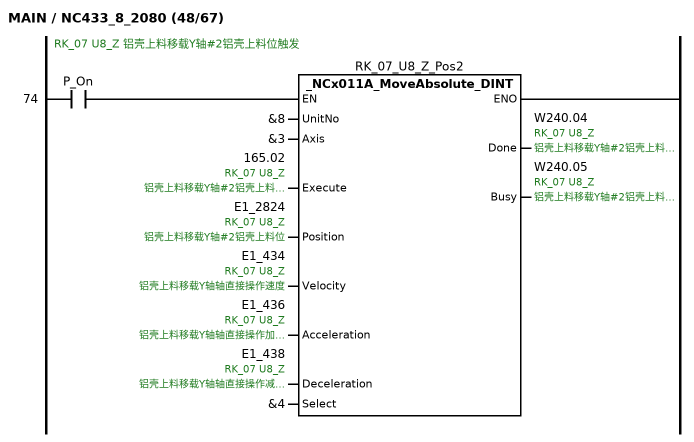
; [picture p312: MAIN / NC433_8_2080, rungs 74-74]
; rung 74: RK_07 U8_Z 铝壳上料移载Y轴#2铝壳上料位触发
LD P_On
CALL RK_07_U8_Z_Pos2 : _NCx011A_MoveAbsolute_DINT (UnitNo := &8, Axis := &3, Execute := 165.02, Position := E1_2824, Velocity := E1_434, Acceleration := E1_436, Deceleration := E1_438, Select := &4, Done => W240.04, Busy => W240.05)  ; RK_07 U8_Z 铝壳上料移载Y轴#2铝壳上料位触发, RK_07 U8_Z 铝壳上料移载Y轴#2铝壳上料位, RK_07 U8_Z 铝壳上料移载Y轴轴直接操作速度, RK_07 U8_Z 铝壳上料移载Y轴轴直接操作加速时间, RK_07 U8_Z 铝壳上料移载Y轴轴直接操作减速时间, RK_07 U8_Z 铝壳上料移载Y轴#2铝壳上料位完成标志, RK_07 U8_Z 铝壳上料移载Y轴#2铝壳上料位忙标志

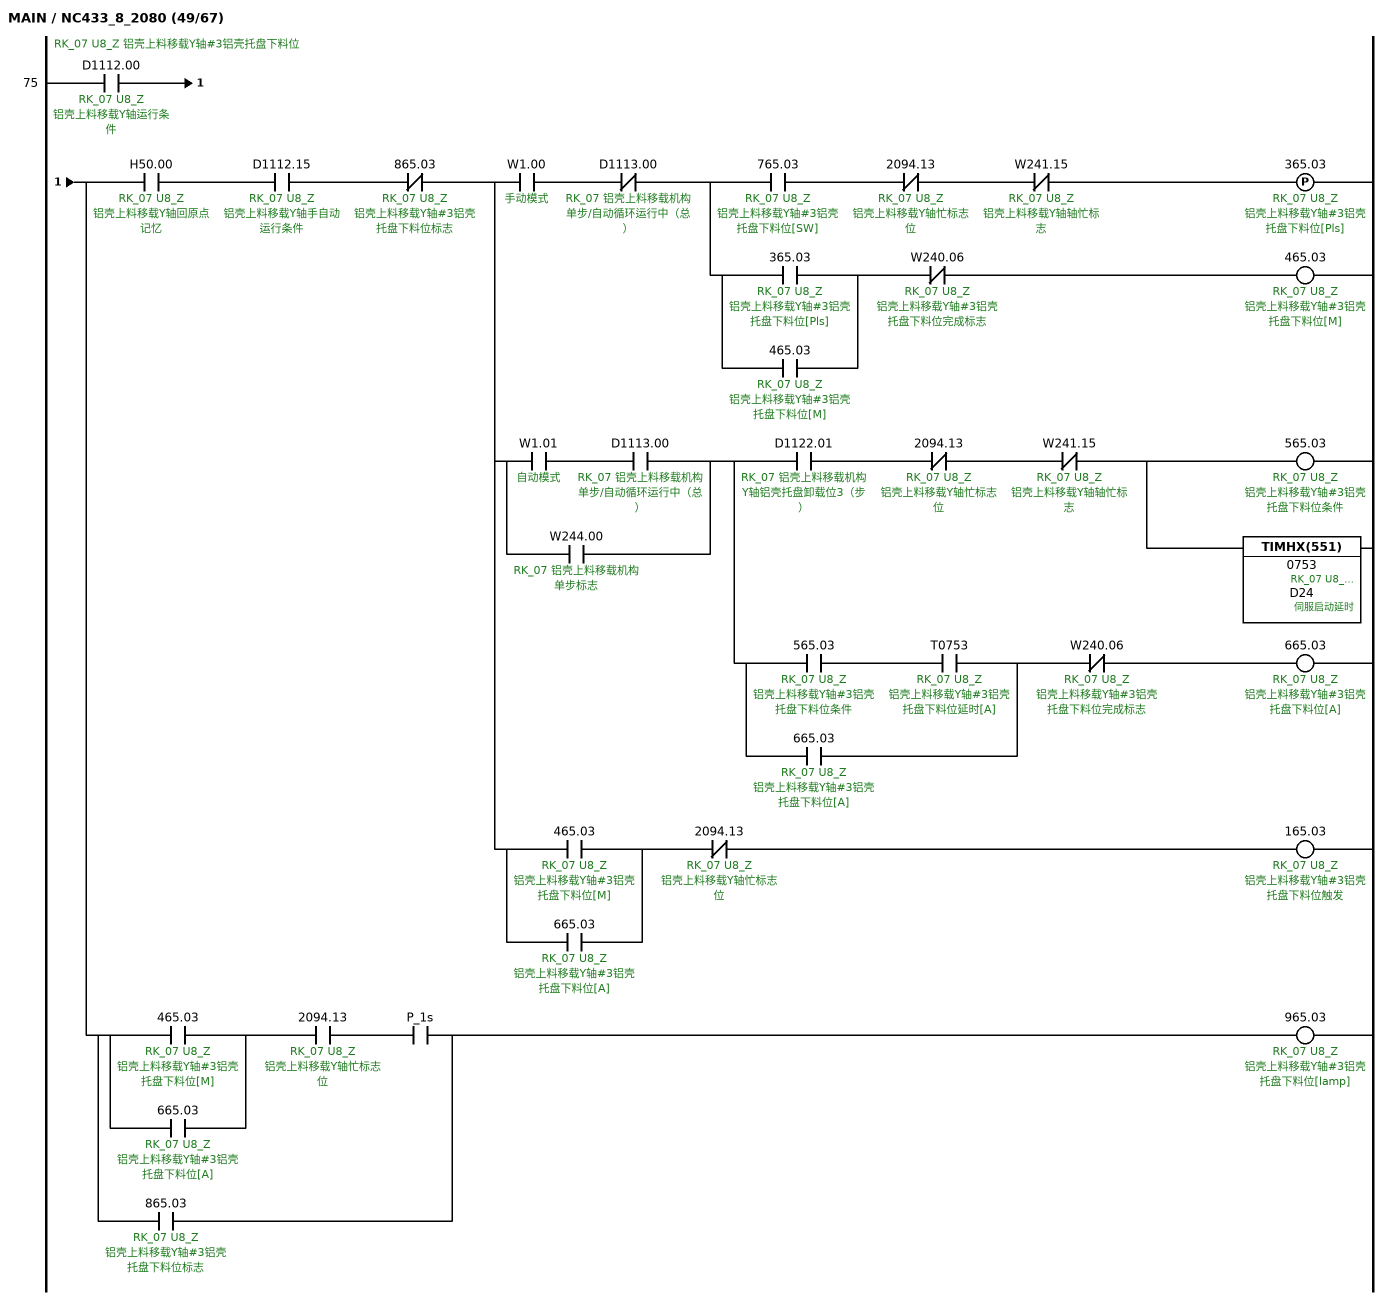
; rung 75: RK_07 U8_Z 铝壳上料移载Y轴#3铝壳托盘下料位
LD D1112.00  ; RK_07 U8_Z 铝壳上料移载Y轴运行条件
OUT TR0
AND H50.00  ; RK_07 U8_Z 铝壳上料移载Y轴回原点记忆
AND D1112.15  ; RK_07 U8_Z 铝壳上料移载Y轴手自动运行条件
ANDNOT 865.03  ; RK_07 U8_Z 铝壳上料移载Y轴#3铝壳托盘下料位标志
OUT TR1
AND W1.00  ; 手动模式
ANDNOT D1113.00  ; RK_07 铝壳上料移载机构单步/自动循环运行中（总）
OUT TR2
AND 765.03  ; RK_07 U8_Z 铝壳上料移载Y轴#3铝壳托盘下料位[SW]
ANDNOT 2094.13  ; RK_07 U8_Z 铝壳上料移载Y轴忙标志位
ANDNOT W241.15  ; RK_07 U8_Z 铝壳上料移载Y轴轴忙标志
DIFU(013) 365.03  ; RK_07 U8_Z 铝壳上料移载Y轴#3铝壳托盘下料位[Pls]
LD TR2
LD 365.03  ; RK_07 U8_Z 铝壳上料移载Y轴#3铝壳托盘下料位[Pls]
OR 465.03  ; RK_07 U8_Z 铝壳上料移载Y轴#3铝壳托盘下料位[M]
ANDLD
ANDNOT W240.06  ; RK_07 U8_Z 铝壳上料移载Y轴#3铝壳托盘下料位完成标志
OUT 465.03  ; RK_07 U8_Z 铝壳上料移载Y轴#3铝壳托盘下料位[M]
LD TR1
LD W1.01  ; 自动模式
AND D1113.00  ; RK_07 铝壳上料移载机构单步/自动循环运行中（总）
OR W244.00  ; RK_07 铝壳上料移载机构单步标志
ANDLD
OUT TR2
AND D1122.01  ; RK_07 铝壳上料移载机构Y轴铝壳托盘卸载位3（步）
ANDNOT 2094.13  ; RK_07 U8_Z 铝壳上料移载Y轴忙标志位
ANDNOT W241.15  ; RK_07 U8_Z 铝壳上料移载Y轴轴忙标志
OUT 565.03  ; RK_07 U8_Z 铝壳上料移载Y轴#3铝壳托盘下料位条件
TIMHX(551) 0753 D24  ; 伺服启动延时, RK_07 U8_Z 铝壳上料移载Y轴#3铝壳托盘下料位延时[A]
LD TR2
LD 565.03  ; RK_07 U8_Z 铝壳上料移载Y轴#3铝壳托盘下料位条件
AND T0753  ; RK_07 U8_Z 铝壳上料移载Y轴#3铝壳托盘下料位延时[A]
OR 665.03  ; RK_07 U8_Z 铝壳上料移载Y轴#3铝壳托盘下料位[A]
ANDLD
ANDNOT W240.06  ; RK_07 U8_Z 铝壳上料移载Y轴#3铝壳托盘下料位完成标志
OUT 665.03  ; RK_07 U8_Z 铝壳上料移载Y轴#3铝壳托盘下料位[A]
LD TR1
LD 465.03  ; RK_07 U8_Z 铝壳上料移载Y轴#3铝壳托盘下料位[M]
OR 665.03  ; RK_07 U8_Z 铝壳上料移载Y轴#3铝壳托盘下料位[A]
ANDLD
ANDNOT 2094.13  ; RK_07 U8_Z 铝壳上料移载Y轴忙标志位
OUT 165.03  ; RK_07 U8_Z 铝壳上料移载Y轴#3铝壳托盘下料位触发
LD TR0
LD 465.03  ; RK_07 U8_Z 铝壳上料移载Y轴#3铝壳托盘下料位[M]
OR 665.03  ; RK_07 U8_Z 铝壳上料移载Y轴#3铝壳托盘下料位[A]
AND 2094.13  ; RK_07 U8_Z 铝壳上料移载Y轴忙标志位
AND P_1s
OR 865.03  ; RK_07 U8_Z 铝壳上料移载Y轴#3铝壳托盘下料位标志
ANDLD
OUT 965.03  ; RK_07 U8_Z 铝壳上料移载Y轴#3铝壳托盘下料位[lamp]

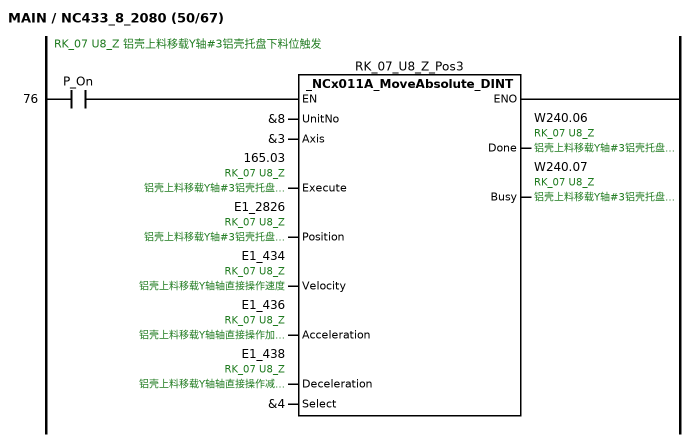
; rung 76: RK_07 U8_Z 铝壳上料移载Y轴#3铝壳托盘下料位触发
LD P_On
CALL RK_07_U8_Z_Pos3 : _NCx011A_MoveAbsolute_DINT (UnitNo := &8, Axis := &3, Execute := 165.03, Position := E1_2826, Velocity := E1_434, Acceleration := E1_436, Deceleration := E1_438, Select := &4, Done => W240.06, Busy => W240.07)  ; RK_07 U8_Z 铝壳上料移载Y轴#3铝壳托盘下料位触发, RK_07 U8_Z 铝壳上料移载Y轴#3铝壳托盘下料位, RK_07 U8_Z 铝壳上料移载Y轴轴直接操作速度, RK_07 U8_Z 铝壳上料移载Y轴轴直接操作加速时间, RK_07 U8_Z 铝壳上料移载Y轴轴直接操作减速时间, RK_07 U8_Z 铝壳上料移载Y轴#3铝壳托盘下料位完成标志, RK_07 U8_Z 铝壳上料移载Y轴#3铝壳托盘下料位忙标志

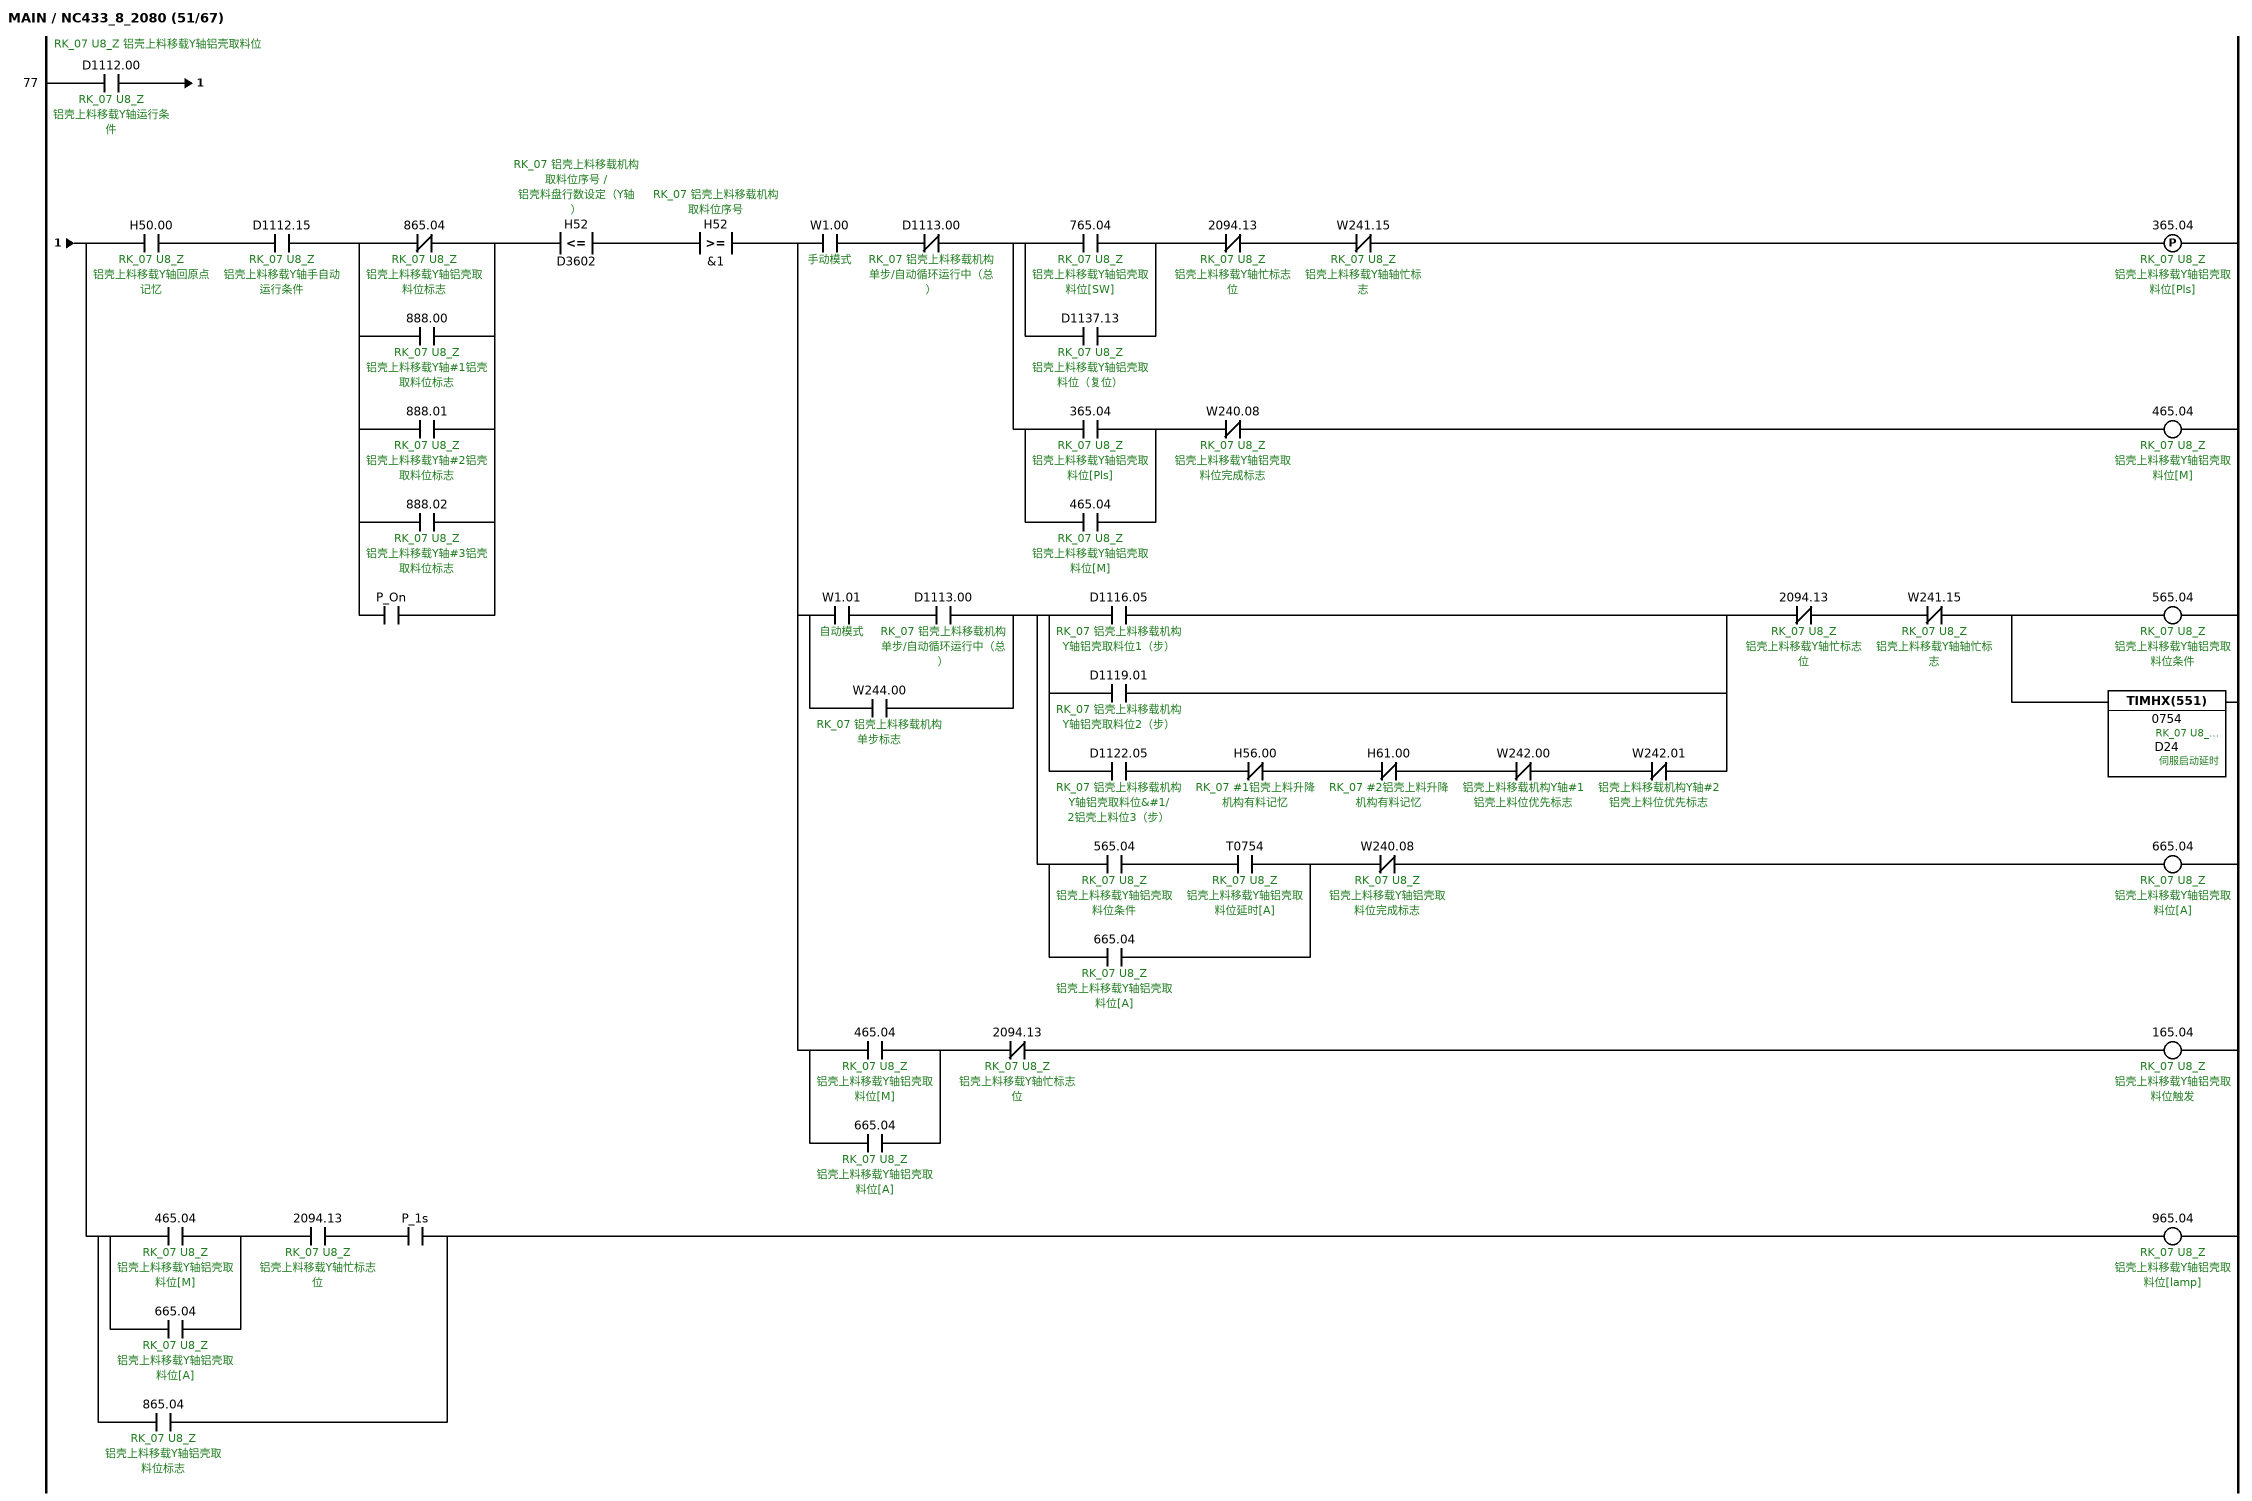
; rung 77: RK_07 U8_Z 铝壳上料移载Y轴铝壳取料位
LD D1112.00  ; RK_07 U8_Z 铝壳上料移载Y轴运行条件
OUT TR0
AND H50.00  ; RK_07 U8_Z 铝壳上料移载Y轴回原点记忆
AND D1112.15  ; RK_07 U8_Z 铝壳上料移载Y轴手自动运行条件
LDNOT 865.04  ; RK_07 U8_Z 铝壳上料移载Y轴铝壳取料位标志
OR 888.00  ; RK_07 U8_Z 铝壳上料移载Y轴#1铝壳取料位标志
OR 888.01  ; RK_07 U8_Z 铝壳上料移载Y轴#2铝壳取料位标志
OR 888.02  ; RK_07 U8_Z 铝壳上料移载Y轴#3铝壳取料位标志
OR P_On
ANDLD
AND<=(315) H52 D3602  ; RK_07 铝壳上料移载机构取料位序号, 铝壳料盘行数设定（Y轴）
AND>=(325) H52 &1  ; RK_07 铝壳上料移载机构取料位序号
OUT TR1
AND W1.00  ; 手动模式
ANDNOT D1113.00  ; RK_07 铝壳上料移载机构单步/自动循环运行中（总）
OUT TR2
LD 765.04  ; RK_07 U8_Z 铝壳上料移载Y轴铝壳取料位[SW]
OR D1137.13  ; RK_07 U8_Z 铝壳上料移载Y轴铝壳取料位（复位）
ANDLD
ANDNOT 2094.13  ; RK_07 U8_Z 铝壳上料移载Y轴忙标志位
ANDNOT W241.15  ; RK_07 U8_Z 铝壳上料移载Y轴轴忙标志
DIFU(013) 365.04  ; RK_07 U8_Z 铝壳上料移载Y轴铝壳取料位[Pls]
LD TR2
LD 365.04  ; RK_07 U8_Z 铝壳上料移载Y轴铝壳取料位[Pls]
OR 465.04  ; RK_07 U8_Z 铝壳上料移载Y轴铝壳取料位[M]
ANDLD
ANDNOT W240.08  ; RK_07 U8_Z 铝壳上料移载Y轴铝壳取料位完成标志
OUT 465.04  ; RK_07 U8_Z 铝壳上料移载Y轴铝壳取料位[M]
LD TR1
LD W1.01  ; 自动模式
AND D1113.00  ; RK_07 铝壳上料移载机构单步/自动循环运行中（总）
OR W244.00  ; RK_07 铝壳上料移载机构单步标志
ANDLD
OUT TR2
LD D1116.05  ; RK_07 铝壳上料移载机构Y轴铝壳取料位1（步）
OR D1119.01  ; RK_07 铝壳上料移载机构Y轴铝壳取料位2（步）
LD D1122.05  ; RK_07 铝壳上料移载机构Y轴铝壳取料位&#1/2铝壳上料位3（步）
ANDNOT H56.00  ; RK_07 #1铝壳上料升降机构有料记忆
ANDNOT H61.00  ; RK_07 #2铝壳上料升降机构有料记忆
ANDNOT W242.00  ; 铝壳上料移载机构Y轴#1铝壳上料位优先标志
ANDNOT W242.01  ; 铝壳上料移载机构Y轴#2铝壳上料位优先标志
ORLD
ANDLD
ANDNOT 2094.13  ; RK_07 U8_Z 铝壳上料移载Y轴忙标志位
ANDNOT W241.15  ; RK_07 U8_Z 铝壳上料移载Y轴轴忙标志
OUT 565.04  ; RK_07 U8_Z 铝壳上料移载Y轴铝壳取料位条件
TIMHX(551) 0754 D24  ; 伺服启动延时, RK_07 U8_Z 铝壳上料移载Y轴铝壳取料位延时[A]
LD TR2
LD 565.04  ; RK_07 U8_Z 铝壳上料移载Y轴铝壳取料位条件
AND T0754  ; RK_07 U8_Z 铝壳上料移载Y轴铝壳取料位延时[A]
OR 665.04  ; RK_07 U8_Z 铝壳上料移载Y轴铝壳取料位[A]
ANDLD
ANDNOT W240.08  ; RK_07 U8_Z 铝壳上料移载Y轴铝壳取料位完成标志
OUT 665.04  ; RK_07 U8_Z 铝壳上料移载Y轴铝壳取料位[A]
LD TR1
LD 465.04  ; RK_07 U8_Z 铝壳上料移载Y轴铝壳取料位[M]
OR 665.04  ; RK_07 U8_Z 铝壳上料移载Y轴铝壳取料位[A]
ANDLD
ANDNOT 2094.13  ; RK_07 U8_Z 铝壳上料移载Y轴忙标志位
OUT 165.04  ; RK_07 U8_Z 铝壳上料移载Y轴铝壳取料位触发
LD TR0
LD 465.04  ; RK_07 U8_Z 铝壳上料移载Y轴铝壳取料位[M]
OR 665.04  ; RK_07 U8_Z 铝壳上料移载Y轴铝壳取料位[A]
AND 2094.13  ; RK_07 U8_Z 铝壳上料移载Y轴忙标志位
AND P_1s
OR 865.04  ; RK_07 U8_Z 铝壳上料移载Y轴铝壳取料位标志
ANDLD
OUT 965.04  ; RK_07 U8_Z 铝壳上料移载Y轴铝壳取料位[lamp]

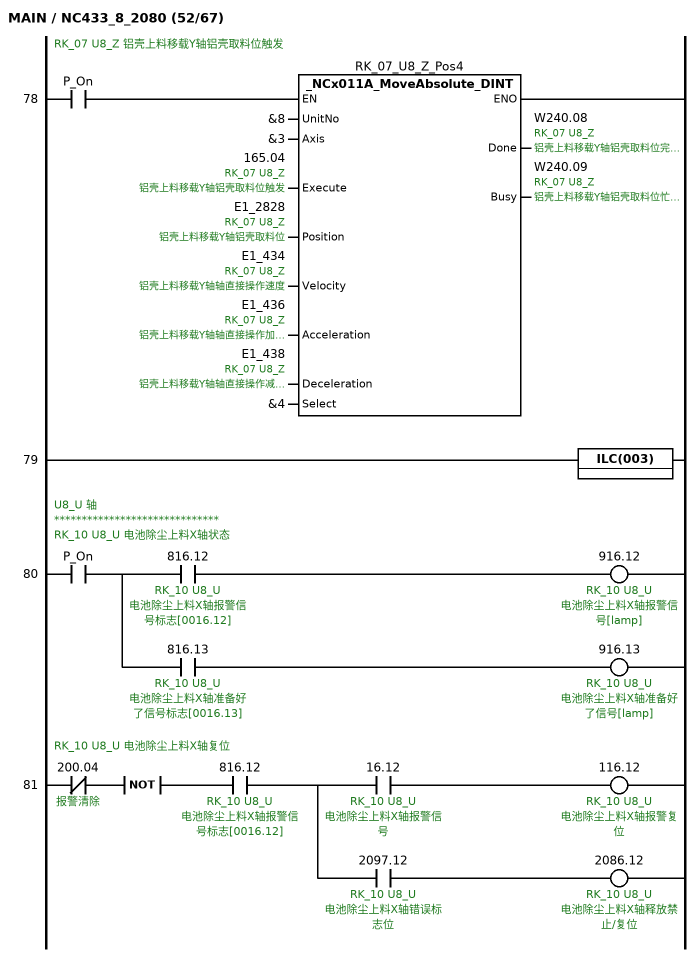
; rung 78: RK_07 U8_Z 铝壳上料移载Y轴铝壳取料位触发
LD P_On
CALL RK_07_U8_Z_Pos4 : _NCx011A_MoveAbsolute_DINT (UnitNo := &8, Axis := &3, Execute := 165.04, Position := E1_2828, Velocity := E1_434, Acceleration := E1_436, Deceleration := E1_438, Select := &4, Done => W240.08, Busy => W240.09)  ; RK_07 U8_Z 铝壳上料移载Y轴铝壳取料位触发, RK_07 U8_Z 铝壳上料移载Y轴铝壳取料位, RK_07 U8_Z 铝壳上料移载Y轴轴直接操作速度, RK_07 U8_Z 铝壳上料移载Y轴轴直接操作加速时间, RK_07 U8_Z 铝壳上料移载Y轴轴直接操作减速时间, RK_07 U8_Z 铝壳上料移载Y轴铝壳取料位完成标志, RK_07 U8_Z 铝壳上料移载Y轴铝壳取料位忙标志
; rung 79
ILC(003)
; rung 80: U8_U 轴 / ****************************** / RK_10 U8_U 电池除尘上料X轴状态
LD P_On
OUT TR0
AND 816.12  ; RK_10 U8_U 电池除尘上料X轴报警信号标志[0016.12]
OUT 916.12  ; RK_10 U8_U 电池除尘上料X轴报警信号[lamp]
LD TR0
AND 816.13  ; RK_10 U8_U 电池除尘上料X轴准备好了信号标志[0016.13]
OUT 916.13  ; RK_10 U8_U 电池除尘上料X轴准备好了信号[lamp]
; rung 81: RK_10 U8_U 电池除尘上料X轴复位
LDNOT 200.04  ; 报警清除
NOT(520)
AND 816.12  ; RK_10 U8_U 电池除尘上料X轴报警信号标志[0016.12]
OUT TR0
AND 16.12  ; RK_10 U8_U 电池除尘上料X轴报警信号
OUT 116.12  ; RK_10 U8_U 电池除尘上料X轴报警复位
LD TR0
AND 2097.12  ; RK_10 U8_U 电池除尘上料X轴错误标志位
OUT 2086.12  ; RK_10 U8_U 电池除尘上料X轴释放禁止/复位

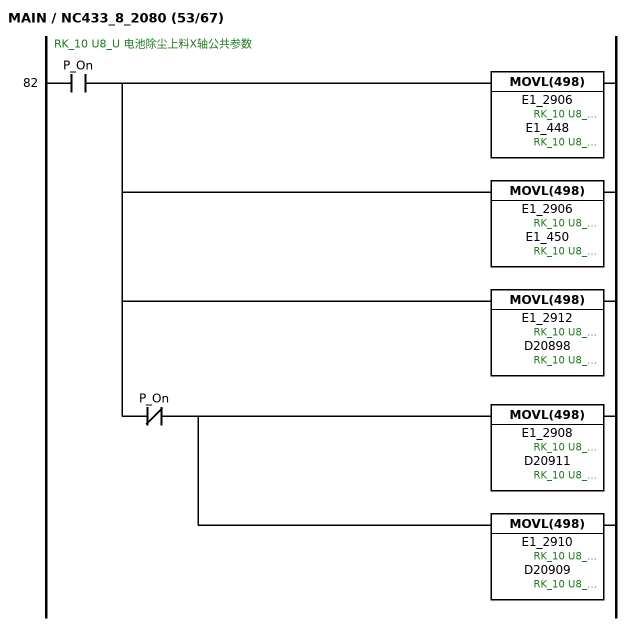
; rung 82: RK_10 U8_U 电池除尘上料X轴公共参数
LD P_On
MOVL(498) E1_2906 E1_448  ; RK_10 U8_U 电池除尘上料X轴轴加减速时间, RK_10 U8_U 电池除尘上料X轴轴直接操作加速时间
MOVL(498) E1_2906 E1_450  ; RK_10 U8_U 电池除尘上料X轴轴加减速时间, RK_10 U8_U 电池除尘上料X轴轴直接操作减速时间
MOVL(498) E1_2912 D20898  ; RK_10 U8_U 电池除尘上料X轴轴原点偏移, RK_10 U8_U 电池除尘上料X轴轴原点补偿值
ANDNOT P_On
MOVL(498) E1_2908 D20911  ; RK_10 U8_U 电池除尘上料X轴轴正软极限, RK_10 U8_U 电池除尘上料X轴轴正软限位
MOVL(498) E1_2910 D20909  ; RK_10 U8_U 电池除尘上料X轴轴负软极限, RK_10 U8_U 电池除尘上料X轴轴负软限位

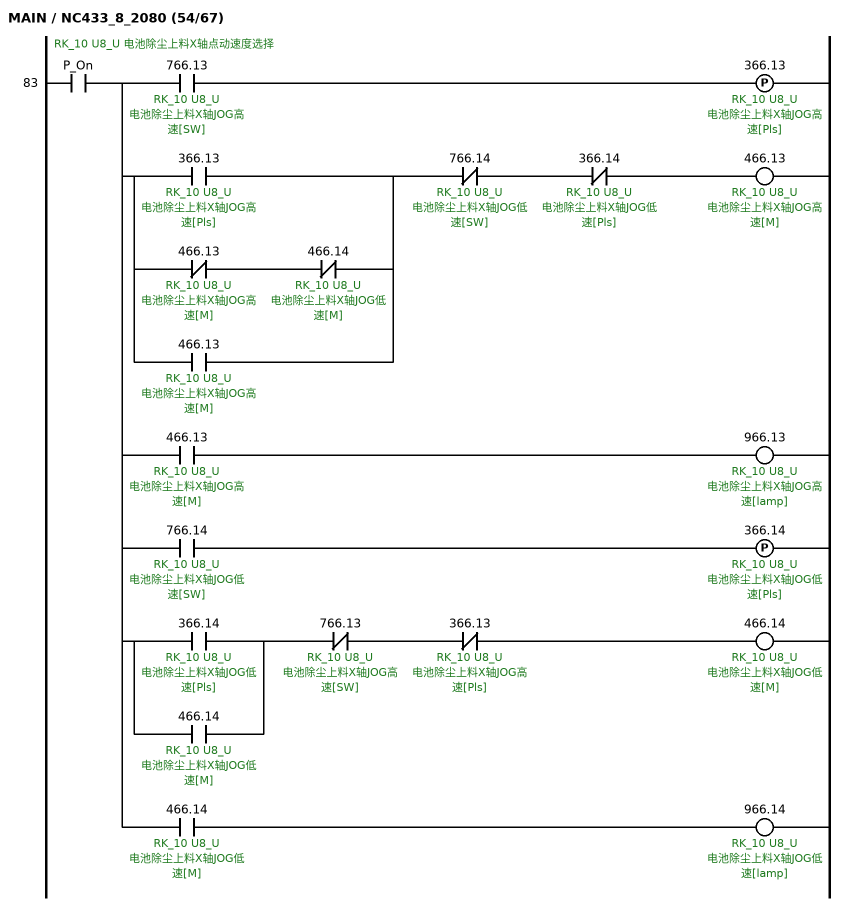
; rung 83: RK_10 U8_U 电池除尘上料X轴点动速度选择
LD P_On
OUT TR0
AND 766.13  ; RK_10 U8_U 电池除尘上料X轴JOG高速[SW]
DIFU(013) 366.13  ; RK_10 U8_U 电池除尘上料X轴JOG高速[Pls]
LD TR0
LD 366.13  ; RK_10 U8_U 电池除尘上料X轴JOG高速[Pls]
LDNOT 466.13  ; RK_10 U8_U 电池除尘上料X轴JOG高速[M]
ANDNOT 466.14  ; RK_10 U8_U 电池除尘上料X轴JOG低速[M]
ORLD
OR 466.13  ; RK_10 U8_U 电池除尘上料X轴JOG高速[M]
ANDLD
ANDNOT 766.14  ; RK_10 U8_U 电池除尘上料X轴JOG低速[SW]
ANDNOT 366.14  ; RK_10 U8_U 电池除尘上料X轴JOG低速[Pls]
OUT 466.13  ; RK_10 U8_U 电池除尘上料X轴JOG高速[M]
LD TR0
AND 466.13  ; RK_10 U8_U 电池除尘上料X轴JOG高速[M]
OUT 966.13  ; RK_10 U8_U 电池除尘上料X轴JOG高速[lamp]
LD TR0
AND 766.14  ; RK_10 U8_U 电池除尘上料X轴JOG低速[SW]
DIFU(013) 366.14  ; RK_10 U8_U 电池除尘上料X轴JOG低速[Pls]
LD TR0
LD 366.14  ; RK_10 U8_U 电池除尘上料X轴JOG低速[Pls]
OR 466.14  ; RK_10 U8_U 电池除尘上料X轴JOG低速[M]
ANDLD
ANDNOT 766.13  ; RK_10 U8_U 电池除尘上料X轴JOG高速[SW]
ANDNOT 366.13  ; RK_10 U8_U 电池除尘上料X轴JOG高速[Pls]
OUT 466.14  ; RK_10 U8_U 电池除尘上料X轴JOG低速[M]
LD TR0
AND 466.14  ; RK_10 U8_U 电池除尘上料X轴JOG低速[M]
OUT 966.14  ; RK_10 U8_U 电池除尘上料X轴JOG低速[lamp]

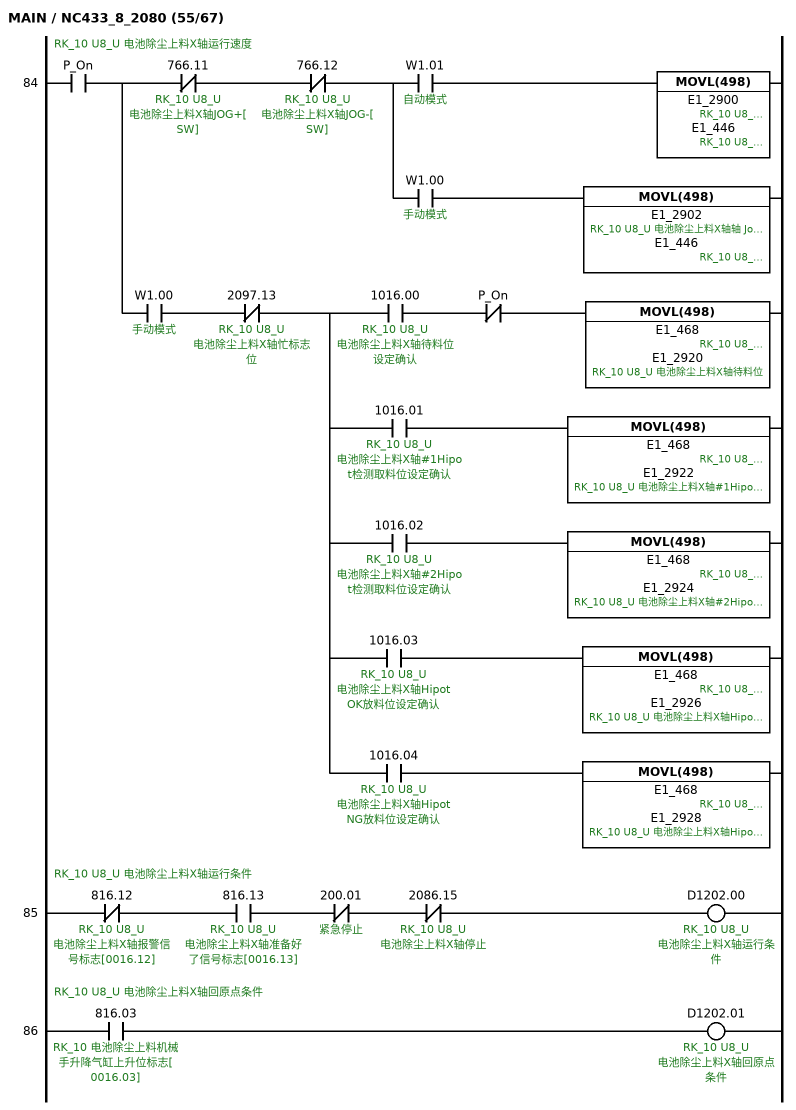
; rung 84: RK_10 U8_U 电池除尘上料X轴运行速度
LD P_On
OUT TR0
ANDNOT 766.11  ; RK_10 U8_U 电池除尘上料X轴JOG+[SW]
ANDNOT 766.12  ; RK_10 U8_U 电池除尘上料X轴JOG-[SW]
OUT TR1
AND W1.01  ; 自动模式
MOVL(498) E1_2900 E1_446  ; RK_10 U8_U 电池除尘上料X轴轴自动速度, RK_10 U8_U 电池除尘上料X轴轴直接操作速度
LD TR1
AND W1.00  ; 手动模式
MOVL(498) E1_2902 E1_446  ; RK_10 U8_U 电池除尘上料X轴轴 Jog 高速, RK_10 U8_U 电池除尘上料X轴轴直接操作速度
LD TR0
AND W1.00  ; 手动模式
ANDNOT 2097.13  ; RK_10 U8_U 电池除尘上料X轴忙标志位
OUT TR0
AND 1016.00  ; RK_10 U8_U 电池除尘上料X轴待料位设定确认
ANDNOT P_On
MOVL(498) E1_468 E1_2920  ; RK_10 U8_U 电池除尘上料X轴轴当前位置, RK_10 U8_U 电池除尘上料X轴待料位
LD TR0
AND 1016.01  ; RK_10 U8_U 电池除尘上料X轴#1Hipot检测取料位设定确认
MOVL(498) E1_468 E1_2922  ; RK_10 U8_U 电池除尘上料X轴轴当前位置, RK_10 U8_U 电池除尘上料X轴#1Hipot检测取料位
LD TR0
AND 1016.02  ; RK_10 U8_U 电池除尘上料X轴#2Hipot检测取料位设定确认
MOVL(498) E1_468 E1_2924  ; RK_10 U8_U 电池除尘上料X轴轴当前位置, RK_10 U8_U 电池除尘上料X轴#2Hipot检测取料位
LD TR0
AND 1016.03  ; RK_10 U8_U 电池除尘上料X轴Hipot OK放料位设定确认
MOVL(498) E1_468 E1_2926  ; RK_10 U8_U 电池除尘上料X轴轴当前位置, RK_10 U8_U 电池除尘上料X轴Hipot OK放料位
LD TR0
AND 1016.04  ; RK_10 U8_U 电池除尘上料X轴Hipot NG放料位设定确认
MOVL(498) E1_468 E1_2928  ; RK_10 U8_U 电池除尘上料X轴轴当前位置, RK_10 U8_U 电池除尘上料X轴Hipot NG放料位
; rung 85: RK_10 U8_U 电池除尘上料X轴运行条件
LDNOT 816.12  ; RK_10 U8_U 电池除尘上料X轴报警信号标志[0016.12]
AND 816.13  ; RK_10 U8_U 电池除尘上料X轴准备好了信号标志[0016.13]
ANDNOT 200.01  ; 紧急停止
ANDNOT 2086.15  ; RK_10 U8_U 电池除尘上料X轴停止
OUT D1202.00  ; RK_10 U8_U 电池除尘上料X轴运行条件
; rung 86: RK_10 U8_U 电池除尘上料X轴回原点条件
LD 816.03  ; RK_10 电池除尘上料机械手升降气缸上升位标志[0016.03]
OUT D1202.01  ; RK_10 U8_U 电池除尘上料X轴回原点条件

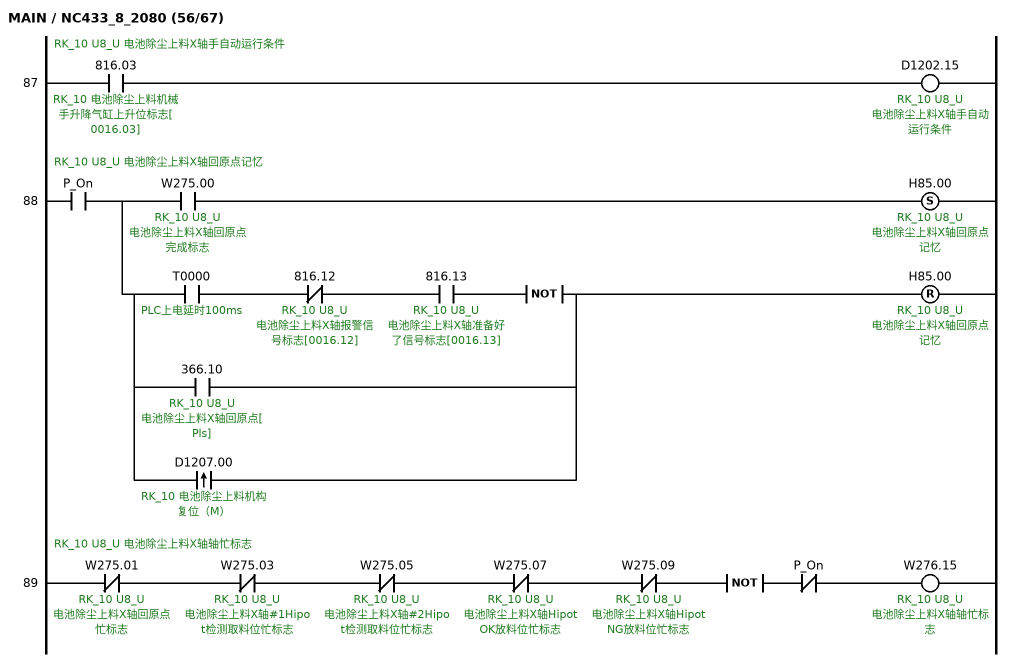
; rung 87: RK_10 U8_U 电池除尘上料X轴手自动运行条件
LD 816.03  ; RK_10 电池除尘上料机械手升降气缸上升位标志[0016.03]
OUT D1202.15  ; RK_10 U8_U 电池除尘上料X轴手自动运行条件
; rung 88: RK_10 U8_U 电池除尘上料X轴回原点记忆
LD P_On
OUT TR0
AND W275.00  ; RK_10 U8_U 电池除尘上料X轴回原点完成标志
SET H85.00  ; RK_10 U8_U 电池除尘上料X轴回原点记忆
LD TR0
LD T0000  ; PLC上电延时100ms
ANDNOT 816.12  ; RK_10 U8_U 电池除尘上料X轴报警信号标志[0016.12]
AND 816.13  ; RK_10 U8_U 电池除尘上料X轴准备好了信号标志[0016.13]
NOT(520)
OR 366.10  ; RK_10 U8_U 电池除尘上料X轴回原点[Pls]
@OR D1207.00  ; RK_10 电池除尘上料机构复位（M）
ANDLD
RSET H85.00  ; RK_10 U8_U 电池除尘上料X轴回原点记忆
; rung 89: RK_10 U8_U 电池除尘上料X轴轴忙标志
LDNOT W275.01  ; RK_10 U8_U 电池除尘上料X轴回原点忙标志
ANDNOT W275.03  ; RK_10 U8_U 电池除尘上料X轴#1Hipot检测取料位忙标志
ANDNOT W275.05  ; RK_10 U8_U 电池除尘上料X轴#2Hipot检测取料位忙标志
ANDNOT W275.07  ; RK_10 U8_U 电池除尘上料X轴Hipot OK放料位忙标志
ANDNOT W275.09  ; RK_10 U8_U 电池除尘上料X轴Hipot NG放料位忙标志
NOT(520)
ANDNOT P_On
OUT W276.15  ; RK_10 U8_U 电池除尘上料X轴轴忙标志

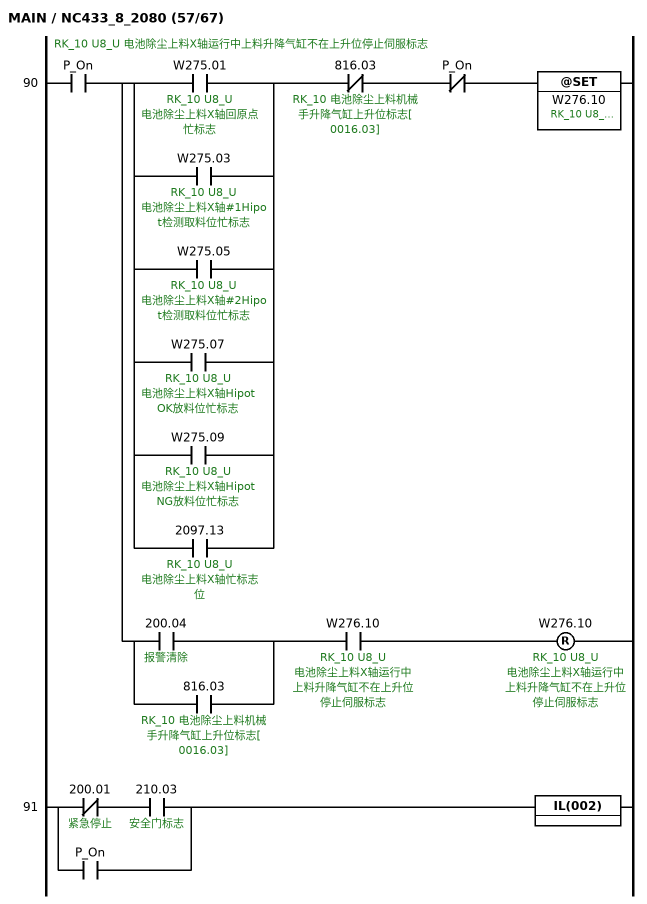
; rung 90: RK_10 U8_U 电池除尘上料X轴运行中上料升降气缸不在上升位停止伺服标志
LD P_On
OUT TR0
LD W275.01  ; RK_10 U8_U 电池除尘上料X轴回原点忙标志
OR W275.03  ; RK_10 U8_U 电池除尘上料X轴#1Hipot检测取料位忙标志
OR W275.05  ; RK_10 U8_U 电池除尘上料X轴#2Hipot检测取料位忙标志
OR W275.07  ; RK_10 U8_U 电池除尘上料X轴Hipot OK放料位忙标志
OR W275.09  ; RK_10 U8_U 电池除尘上料X轴Hipot NG放料位忙标志
OR 2097.13  ; RK_10 U8_U 电池除尘上料X轴忙标志位
ANDLD
ANDNOT 816.03  ; RK_10 电池除尘上料机械手升降气缸上升位标志[0016.03]
ANDNOT P_On
@SET W276.10  ; RK_10 U8_U 电池除尘上料X轴运行中上料升降气缸不在上升位停止伺服标志  // 增加相应报警信息
LD TR0
LD 200.04  ; 报警清除
OR 816.03  ; RK_10 电池除尘上料机械手升降气缸上升位标志[0016.03]
ANDLD
AND W276.10  ; RK_10 U8_U 电池除尘上料X轴运行中上料升降气缸不在上升位停止伺服标志
RSET W276.10  ; RK_10 U8_U 电池除尘上料X轴运行中上料升降气缸不在上升位停止伺服标志
; rung 91
LDNOT 200.01  ; 紧急停止
AND 210.03  ; 安全门标志
OR P_On
IL(002)

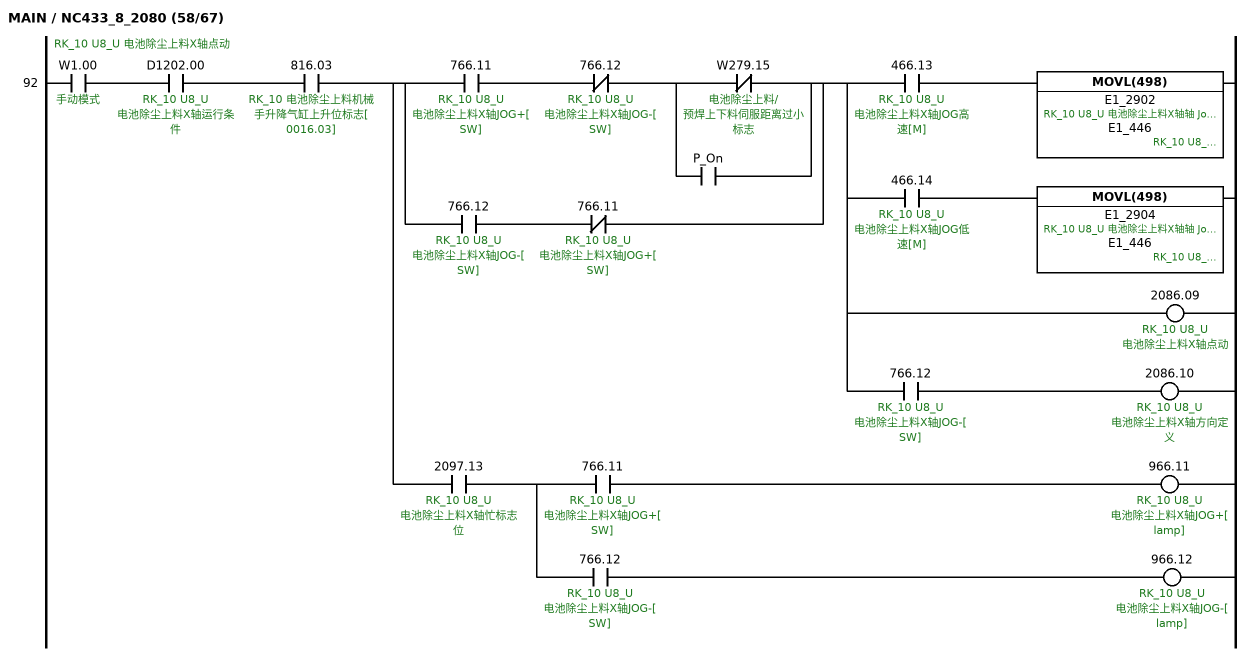
; rung 92: RK_10 U8_U 电池除尘上料X轴点动
LD W1.00  ; 手动模式
AND D1202.00  ; RK_10 U8_U 电池除尘上料X轴运行条件
AND 816.03  ; RK_10 电池除尘上料机械手升降气缸上升位标志[0016.03]
OUT TR0
LD 766.11  ; RK_10 U8_U 电池除尘上料X轴JOG+[SW]
ANDNOT 766.12  ; RK_10 U8_U 电池除尘上料X轴JOG-[SW]
LDNOT W279.15  ; 电池除尘上料/预焊上下料伺服距离过小标志
OR P_On
ANDLD
LD 766.12  ; RK_10 U8_U 电池除尘上料X轴JOG-[SW]
ANDNOT 766.11  ; RK_10 U8_U 电池除尘上料X轴JOG+[SW]
ORLD
ANDLD
OUT TR1
AND 466.13  ; RK_10 U8_U 电池除尘上料X轴JOG高速[M]
MOVL(498) E1_2902 E1_446  ; RK_10 U8_U 电池除尘上料X轴轴 Jog 高速, RK_10 U8_U 电池除尘上料X轴轴直接操作速度
LD TR1
AND 466.14  ; RK_10 U8_U 电池除尘上料X轴JOG低速[M]
MOVL(498) E1_2904 E1_446  ; RK_10 U8_U 电池除尘上料X轴轴 Jog 低速, RK_10 U8_U 电池除尘上料X轴轴直接操作速度
LD TR1
OUT 2086.09  ; RK_10 U8_U 电池除尘上料X轴点动
AND 766.12  ; RK_10 U8_U 电池除尘上料X轴JOG-[SW]
OUT 2086.10  ; RK_10 U8_U 电池除尘上料X轴方向定义
LD TR0
AND 2097.13  ; RK_10 U8_U 电池除尘上料X轴忙标志位
OUT TR0
AND 766.11  ; RK_10 U8_U 电池除尘上料X轴JOG+[SW]
OUT 966.11  ; RK_10 U8_U 电池除尘上料X轴JOG+[lamp]
LD TR0
AND 766.12  ; RK_10 U8_U 电池除尘上料X轴JOG-[SW]
OUT 966.12  ; RK_10 U8_U 电池除尘上料X轴JOG-[lamp]

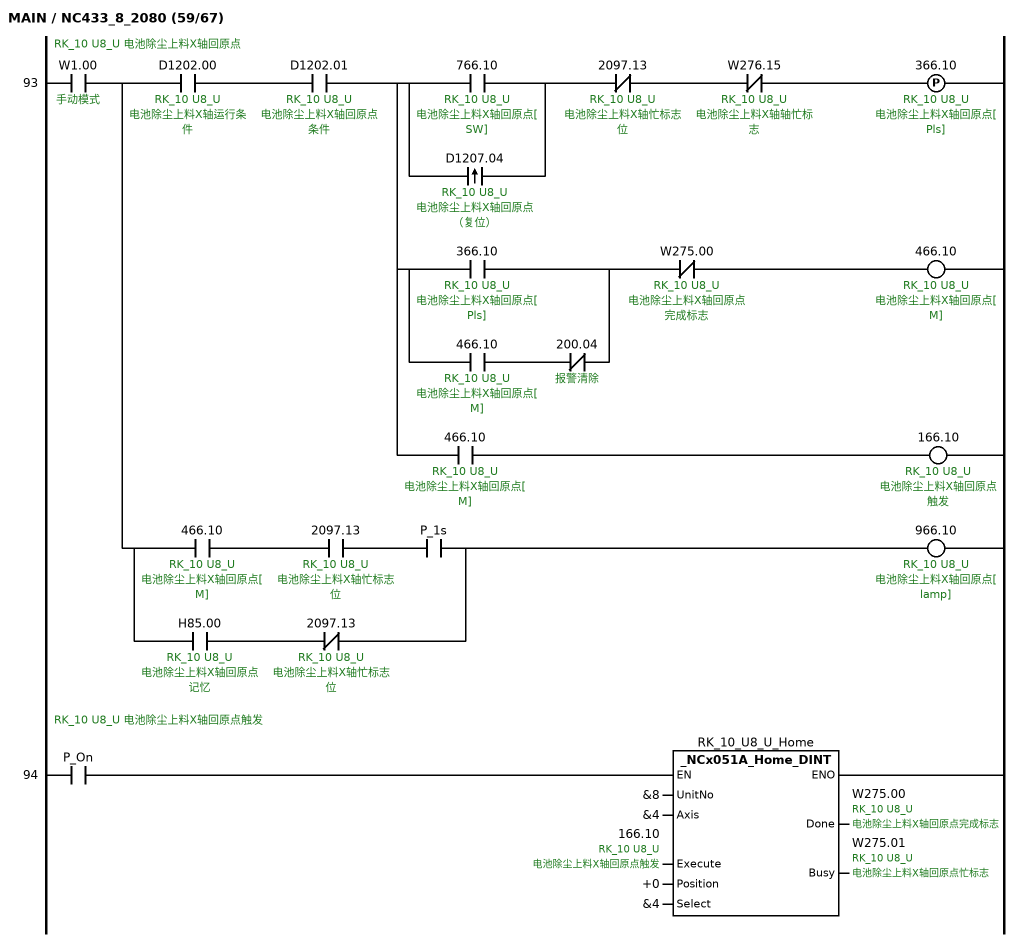
; rung 93: RK_10 U8_U 电池除尘上料X轴回原点
LD W1.00  ; 手动模式
OUT TR0
AND D1202.00  ; RK_10 U8_U 电池除尘上料X轴运行条件
AND D1202.01  ; RK_10 U8_U 电池除尘上料X轴回原点条件
OUT TR1
LD 766.10  ; RK_10 U8_U 电池除尘上料X轴回原点[SW]
@OR D1207.04  ; RK_10 U8_U 电池除尘上料X轴回原点（复位）
ANDLD
ANDNOT 2097.13  ; RK_10 U8_U 电池除尘上料X轴忙标志位
ANDNOT W276.15  ; RK_10 U8_U 电池除尘上料X轴轴忙标志
DIFU(013) 366.10  ; RK_10 U8_U 电池除尘上料X轴回原点[Pls]
LD TR1
LD 366.10  ; RK_10 U8_U 电池除尘上料X轴回原点[Pls]
LD 466.10  ; RK_10 U8_U 电池除尘上料X轴回原点[M]
ANDNOT 200.04  ; 报警清除
ORLD
ANDLD
ANDNOT W275.00  ; RK_10 U8_U 电池除尘上料X轴回原点完成标志
OUT 466.10  ; RK_10 U8_U 电池除尘上料X轴回原点[M]
LD TR1
AND 466.10  ; RK_10 U8_U 电池除尘上料X轴回原点[M]
OUT 166.10  ; RK_10 U8_U 电池除尘上料X轴回原点触发
LD TR0
LD 466.10  ; RK_10 U8_U 电池除尘上料X轴回原点[M]
AND 2097.13  ; RK_10 U8_U 电池除尘上料X轴忙标志位
AND P_1s
LD H85.00  ; RK_10 U8_U 电池除尘上料X轴回原点记忆
ANDNOT 2097.13  ; RK_10 U8_U 电池除尘上料X轴忙标志位
ORLD
ANDLD
OUT 966.10  ; RK_10 U8_U 电池除尘上料X轴回原点[lamp]
; rung 94: RK_10 U8_U 电池除尘上料X轴回原点触发
LD P_On
CALL RK_10_U8_U_Home : _NCx051A_Home_DINT (UnitNo := &8, Axis := &4, Execute := 166.10, Position := +0, Select := &4, Done => W275.00, Busy => W275.01)  ; RK_10 U8_U 电池除尘上料X轴回原点触发, RK_10 U8_U 电池除尘上料X轴回原点完成标志, RK_10 U8_U 电池除尘上料X轴回原点忙标志

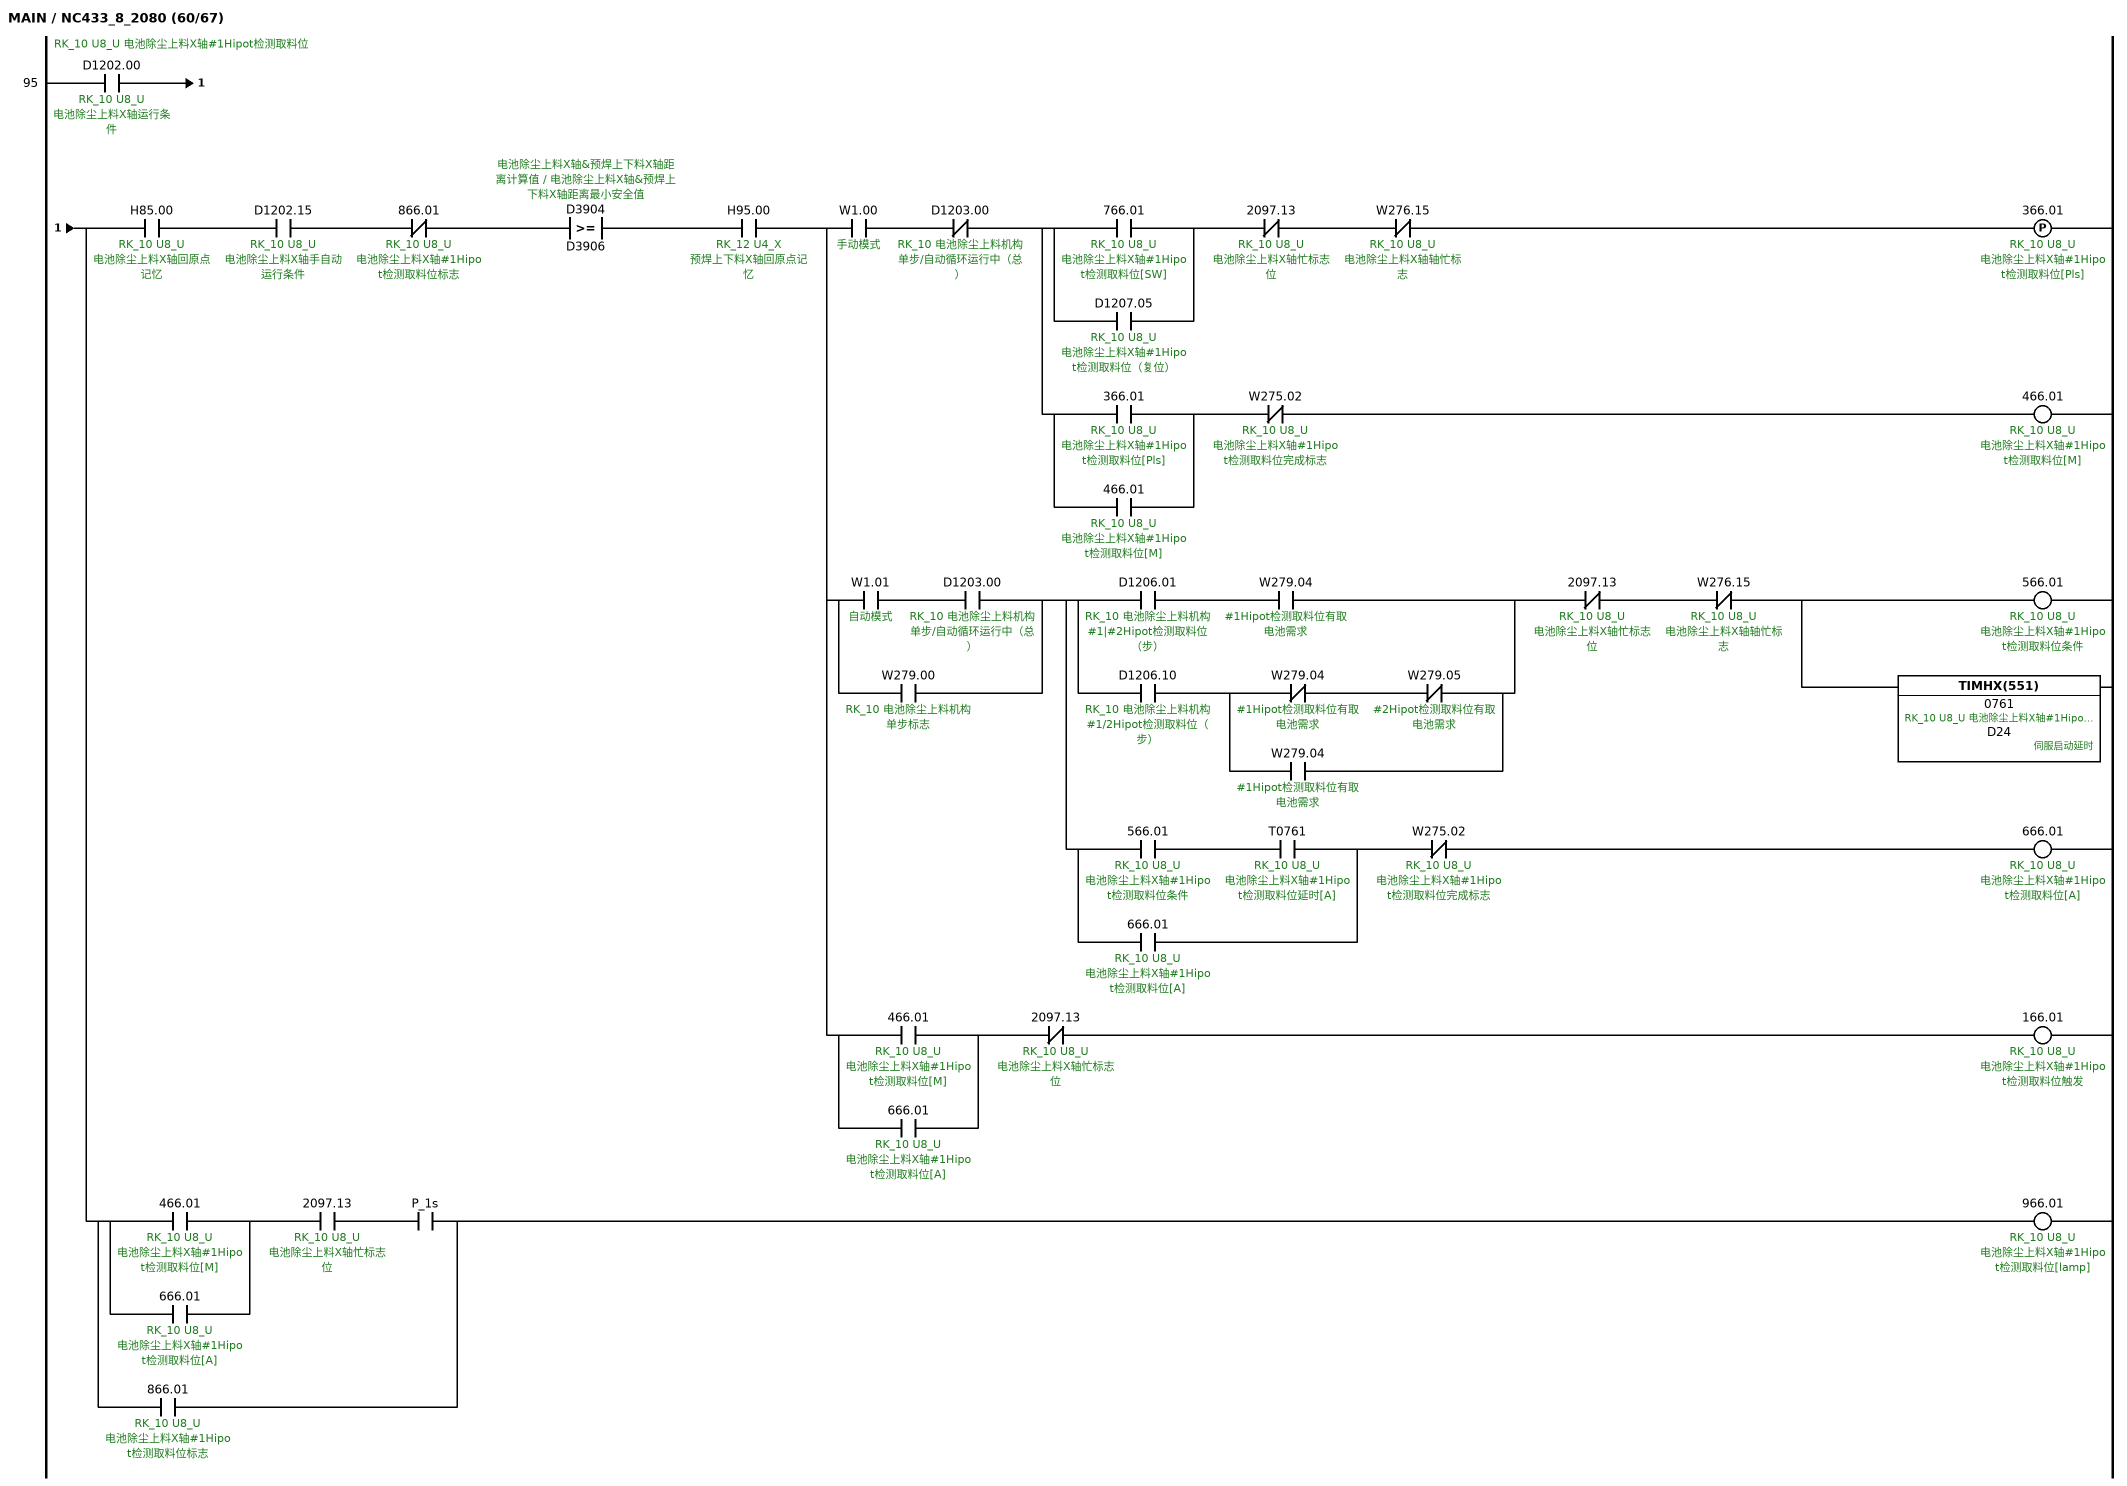
; rung 95: RK_10 U8_U 电池除尘上料X轴#1Hipot检测取料位
LD D1202.00  ; RK_10 U8_U 电池除尘上料X轴运行条件
OUT TR0
AND H85.00  ; RK_10 U8_U 电池除尘上料X轴回原点记忆
AND D1202.15  ; RK_10 U8_U 电池除尘上料X轴手自动运行条件
ANDNOT 866.01  ; RK_10 U8_U 电池除尘上料X轴#1Hipot检测取料位标志
AND>=SL(328) D3904 D3906  ; 电池除尘上料X轴&预焊上下料X轴距离计算值, 电池除尘上料X轴&预焊上下料X轴距离最小安全值
AND H95.00  ; RK_12 U4_X 预焊上下料X轴回原点记忆
OUT TR1
AND W1.00  ; 手动模式
ANDNOT D1203.00  ; RK_10 电池除尘上料机构单步/自动循环运行中（总）
OUT TR2
LD 766.01  ; RK_10 U8_U 电池除尘上料X轴#1Hipot检测取料位[SW]
OR D1207.05  ; RK_10 U8_U 电池除尘上料X轴#1Hipot检测取料位（复位）
ANDLD
ANDNOT 2097.13  ; RK_10 U8_U 电池除尘上料X轴忙标志位
ANDNOT W276.15  ; RK_10 U8_U 电池除尘上料X轴轴忙标志
DIFU(013) 366.01  ; RK_10 U8_U 电池除尘上料X轴#1Hipot检测取料位[Pls]
LD TR2
LD 366.01  ; RK_10 U8_U 电池除尘上料X轴#1Hipot检测取料位[Pls]
OR 466.01  ; RK_10 U8_U 电池除尘上料X轴#1Hipot检测取料位[M]
ANDLD
ANDNOT W275.02  ; RK_10 U8_U 电池除尘上料X轴#1Hipot检测取料位完成标志
OUT 466.01  ; RK_10 U8_U 电池除尘上料X轴#1Hipot检测取料位[M]
LD TR1
LD W1.01  ; 自动模式
AND D1203.00  ; RK_10 电池除尘上料机构单步/自动循环运行中（总）
OR W279.00  ; RK_10 电池除尘上料机构单步标志
ANDLD
OUT TR2
LD D1206.01  ; RK_10 电池除尘上料机构#1|#2Hipot检测取料位（步）
AND W279.04  ; #1Hipot检测取料位有取电池需求
LD D1206.10  ; RK_10 电池除尘上料机构#1/2Hipot检测取料位（步）
LDNOT W279.04  ; #1Hipot检测取料位有取电池需求
ANDNOT W279.05  ; #2Hipot检测取料位有取电池需求
OR W279.04  ; #1Hipot检测取料位有取电池需求
ANDLD
ORLD
ANDLD
ANDNOT 2097.13  ; RK_10 U8_U 电池除尘上料X轴忙标志位
ANDNOT W276.15  ; RK_10 U8_U 电池除尘上料X轴轴忙标志
OUT 566.01  ; RK_10 U8_U 电池除尘上料X轴#1Hipot检测取料位条件
TIMHX(551) 0761 D24  ; 伺服启动延时, RK_10 U8_U 电池除尘上料X轴#1Hipot检测取料位延时[A]
LD TR2
LD 566.01  ; RK_10 U8_U 电池除尘上料X轴#1Hipot检测取料位条件
AND T0761  ; RK_10 U8_U 电池除尘上料X轴#1Hipot检测取料位延时[A]
OR 666.01  ; RK_10 U8_U 电池除尘上料X轴#1Hipot检测取料位[A]
ANDLD
ANDNOT W275.02  ; RK_10 U8_U 电池除尘上料X轴#1Hipot检测取料位完成标志
OUT 666.01  ; RK_10 U8_U 电池除尘上料X轴#1Hipot检测取料位[A]
LD TR1
LD 466.01  ; RK_10 U8_U 电池除尘上料X轴#1Hipot检测取料位[M]
OR 666.01  ; RK_10 U8_U 电池除尘上料X轴#1Hipot检测取料位[A]
ANDLD
ANDNOT 2097.13  ; RK_10 U8_U 电池除尘上料X轴忙标志位
OUT 166.01  ; RK_10 U8_U 电池除尘上料X轴#1Hipot检测取料位触发
LD TR0
LD 466.01  ; RK_10 U8_U 电池除尘上料X轴#1Hipot检测取料位[M]
OR 666.01  ; RK_10 U8_U 电池除尘上料X轴#1Hipot检测取料位[A]
AND 2097.13  ; RK_10 U8_U 电池除尘上料X轴忙标志位
AND P_1s
OR 866.01  ; RK_10 U8_U 电池除尘上料X轴#1Hipot检测取料位标志
ANDLD
OUT 966.01  ; RK_10 U8_U 电池除尘上料X轴#1Hipot检测取料位[lamp]

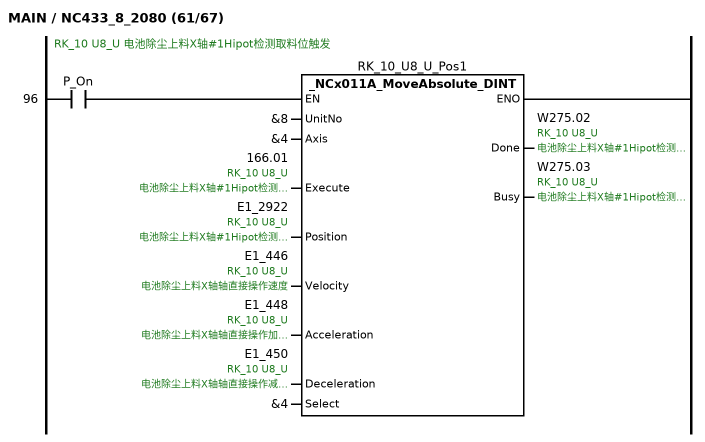
; rung 96: RK_10 U8_U 电池除尘上料X轴#1Hipot检测取料位触发
LD P_On
CALL RK_10_U8_U_Pos1 : _NCx011A_MoveAbsolute_DINT (UnitNo := &8, Axis := &4, Execute := 166.01, Position := E1_2922, Velocity := E1_446, Acceleration := E1_448, Deceleration := E1_450, Select := &4, Done => W275.02, Busy => W275.03)  ; RK_10 U8_U 电池除尘上料X轴#1Hipot检测取料位触发, RK_10 U8_U 电池除尘上料X轴#1Hipot检测取料位, RK_10 U8_U 电池除尘上料X轴轴直接操作速度, RK_10 U8_U 电池除尘上料X轴轴直接操作加速时间, RK_10 U8_U 电池除尘上料X轴轴直接操作减速时间, RK_10 U8_U 电池除尘上料X轴#1Hipot检测取料位完成标志, RK_10 U8_U 电池除尘上料X轴#1Hipot检测取料位忙标志

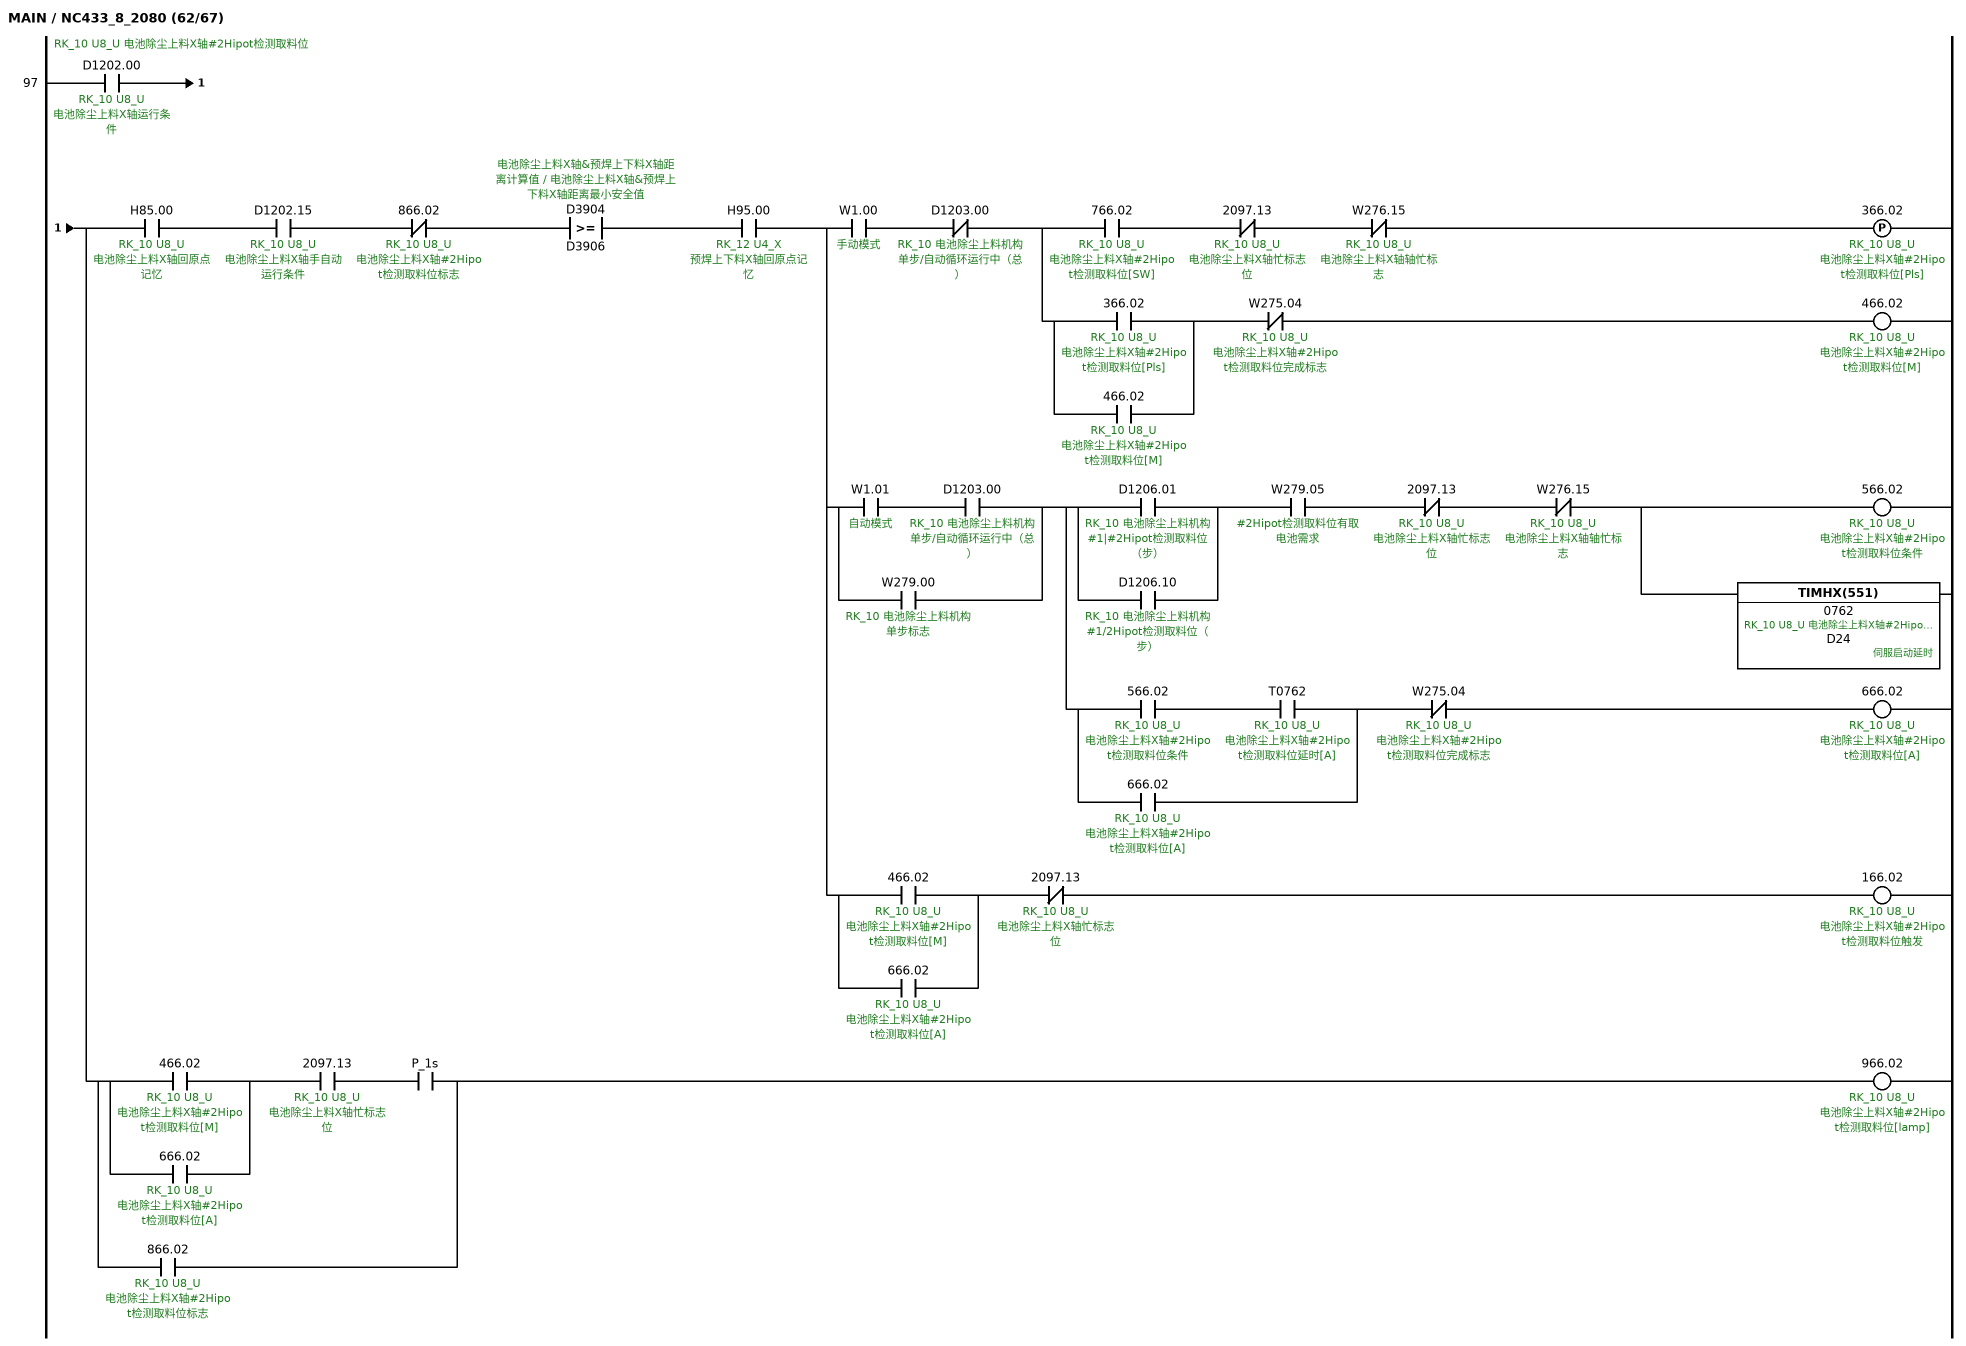
; rung 97: RK_10 U8_U 电池除尘上料X轴#2Hipot检测取料位
LD D1202.00  ; RK_10 U8_U 电池除尘上料X轴运行条件
OUT TR0
AND H85.00  ; RK_10 U8_U 电池除尘上料X轴回原点记忆
AND D1202.15  ; RK_10 U8_U 电池除尘上料X轴手自动运行条件
ANDNOT 866.02  ; RK_10 U8_U 电池除尘上料X轴#2Hipot检测取料位标志
AND>=SL(328) D3904 D3906  ; 电池除尘上料X轴&预焊上下料X轴距离计算值, 电池除尘上料X轴&预焊上下料X轴距离最小安全值
AND H95.00  ; RK_12 U4_X 预焊上下料X轴回原点记忆
OUT TR1
AND W1.00  ; 手动模式
ANDNOT D1203.00  ; RK_10 电池除尘上料机构单步/自动循环运行中（总）
OUT TR2
AND 766.02  ; RK_10 U8_U 电池除尘上料X轴#2Hipot检测取料位[SW]
ANDNOT 2097.13  ; RK_10 U8_U 电池除尘上料X轴忙标志位
ANDNOT W276.15  ; RK_10 U8_U 电池除尘上料X轴轴忙标志
DIFU(013) 366.02  ; RK_10 U8_U 电池除尘上料X轴#2Hipot检测取料位[Pls]
LD TR2
LD 366.02  ; RK_10 U8_U 电池除尘上料X轴#2Hipot检测取料位[Pls]
OR 466.02  ; RK_10 U8_U 电池除尘上料X轴#2Hipot检测取料位[M]
ANDLD
ANDNOT W275.04  ; RK_10 U8_U 电池除尘上料X轴#2Hipot检测取料位完成标志
OUT 466.02  ; RK_10 U8_U 电池除尘上料X轴#2Hipot检测取料位[M]
LD TR1
LD W1.01  ; 自动模式
AND D1203.00  ; RK_10 电池除尘上料机构单步/自动循环运行中（总）
OR W279.00  ; RK_10 电池除尘上料机构单步标志
ANDLD
OUT TR2
LD D1206.01  ; RK_10 电池除尘上料机构#1|#2Hipot检测取料位（步）
OR D1206.10  ; RK_10 电池除尘上料机构#1/2Hipot检测取料位（步）
ANDLD
AND W279.05  ; #2Hipot检测取料位有取电池需求
ANDNOT 2097.13  ; RK_10 U8_U 电池除尘上料X轴忙标志位
ANDNOT W276.15  ; RK_10 U8_U 电池除尘上料X轴轴忙标志
OUT 566.02  ; RK_10 U8_U 电池除尘上料X轴#2Hipot检测取料位条件
TIMHX(551) 0762 D24  ; 伺服启动延时, RK_10 U8_U 电池除尘上料X轴#2Hipot检测取料位延时[A]
LD TR2
LD 566.02  ; RK_10 U8_U 电池除尘上料X轴#2Hipot检测取料位条件
AND T0762  ; RK_10 U8_U 电池除尘上料X轴#2Hipot检测取料位延时[A]
OR 666.02  ; RK_10 U8_U 电池除尘上料X轴#2Hipot检测取料位[A]
ANDLD
ANDNOT W275.04  ; RK_10 U8_U 电池除尘上料X轴#2Hipot检测取料位完成标志
OUT 666.02  ; RK_10 U8_U 电池除尘上料X轴#2Hipot检测取料位[A]
LD TR1
LD 466.02  ; RK_10 U8_U 电池除尘上料X轴#2Hipot检测取料位[M]
OR 666.02  ; RK_10 U8_U 电池除尘上料X轴#2Hipot检测取料位[A]
ANDLD
ANDNOT 2097.13  ; RK_10 U8_U 电池除尘上料X轴忙标志位
OUT 166.02  ; RK_10 U8_U 电池除尘上料X轴#2Hipot检测取料位触发
LD TR0
LD 466.02  ; RK_10 U8_U 电池除尘上料X轴#2Hipot检测取料位[M]
OR 666.02  ; RK_10 U8_U 电池除尘上料X轴#2Hipot检测取料位[A]
AND 2097.13  ; RK_10 U8_U 电池除尘上料X轴忙标志位
AND P_1s
OR 866.02  ; RK_10 U8_U 电池除尘上料X轴#2Hipot检测取料位标志
ANDLD
OUT 966.02  ; RK_10 U8_U 电池除尘上料X轴#2Hipot检测取料位[lamp]

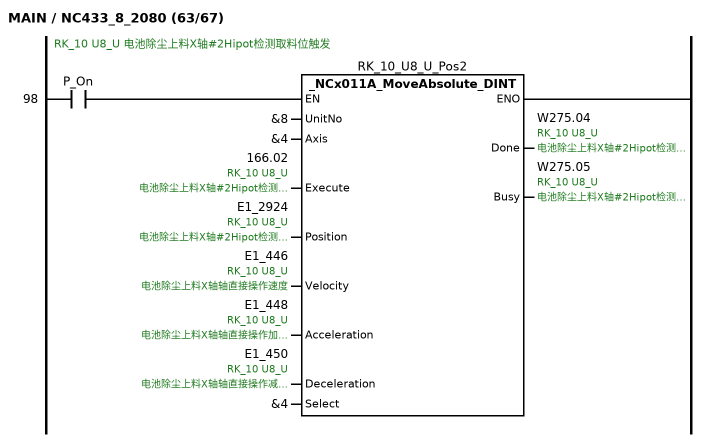
; rung 98: RK_10 U8_U 电池除尘上料X轴#2Hipot检测取料位触发
LD P_On
CALL RK_10_U8_U_Pos2 : _NCx011A_MoveAbsolute_DINT (UnitNo := &8, Axis := &4, Execute := 166.02, Position := E1_2924, Velocity := E1_446, Acceleration := E1_448, Deceleration := E1_450, Select := &4, Done => W275.04, Busy => W275.05)  ; RK_10 U8_U 电池除尘上料X轴#2Hipot检测取料位触发, RK_10 U8_U 电池除尘上料X轴#2Hipot检测取料位, RK_10 U8_U 电池除尘上料X轴轴直接操作速度, RK_10 U8_U 电池除尘上料X轴轴直接操作加速时间, RK_10 U8_U 电池除尘上料X轴轴直接操作减速时间, RK_10 U8_U 电池除尘上料X轴#2Hipot检测取料位完成标志, RK_10 U8_U 电池除尘上料X轴#2Hipot检测取料位忙标志

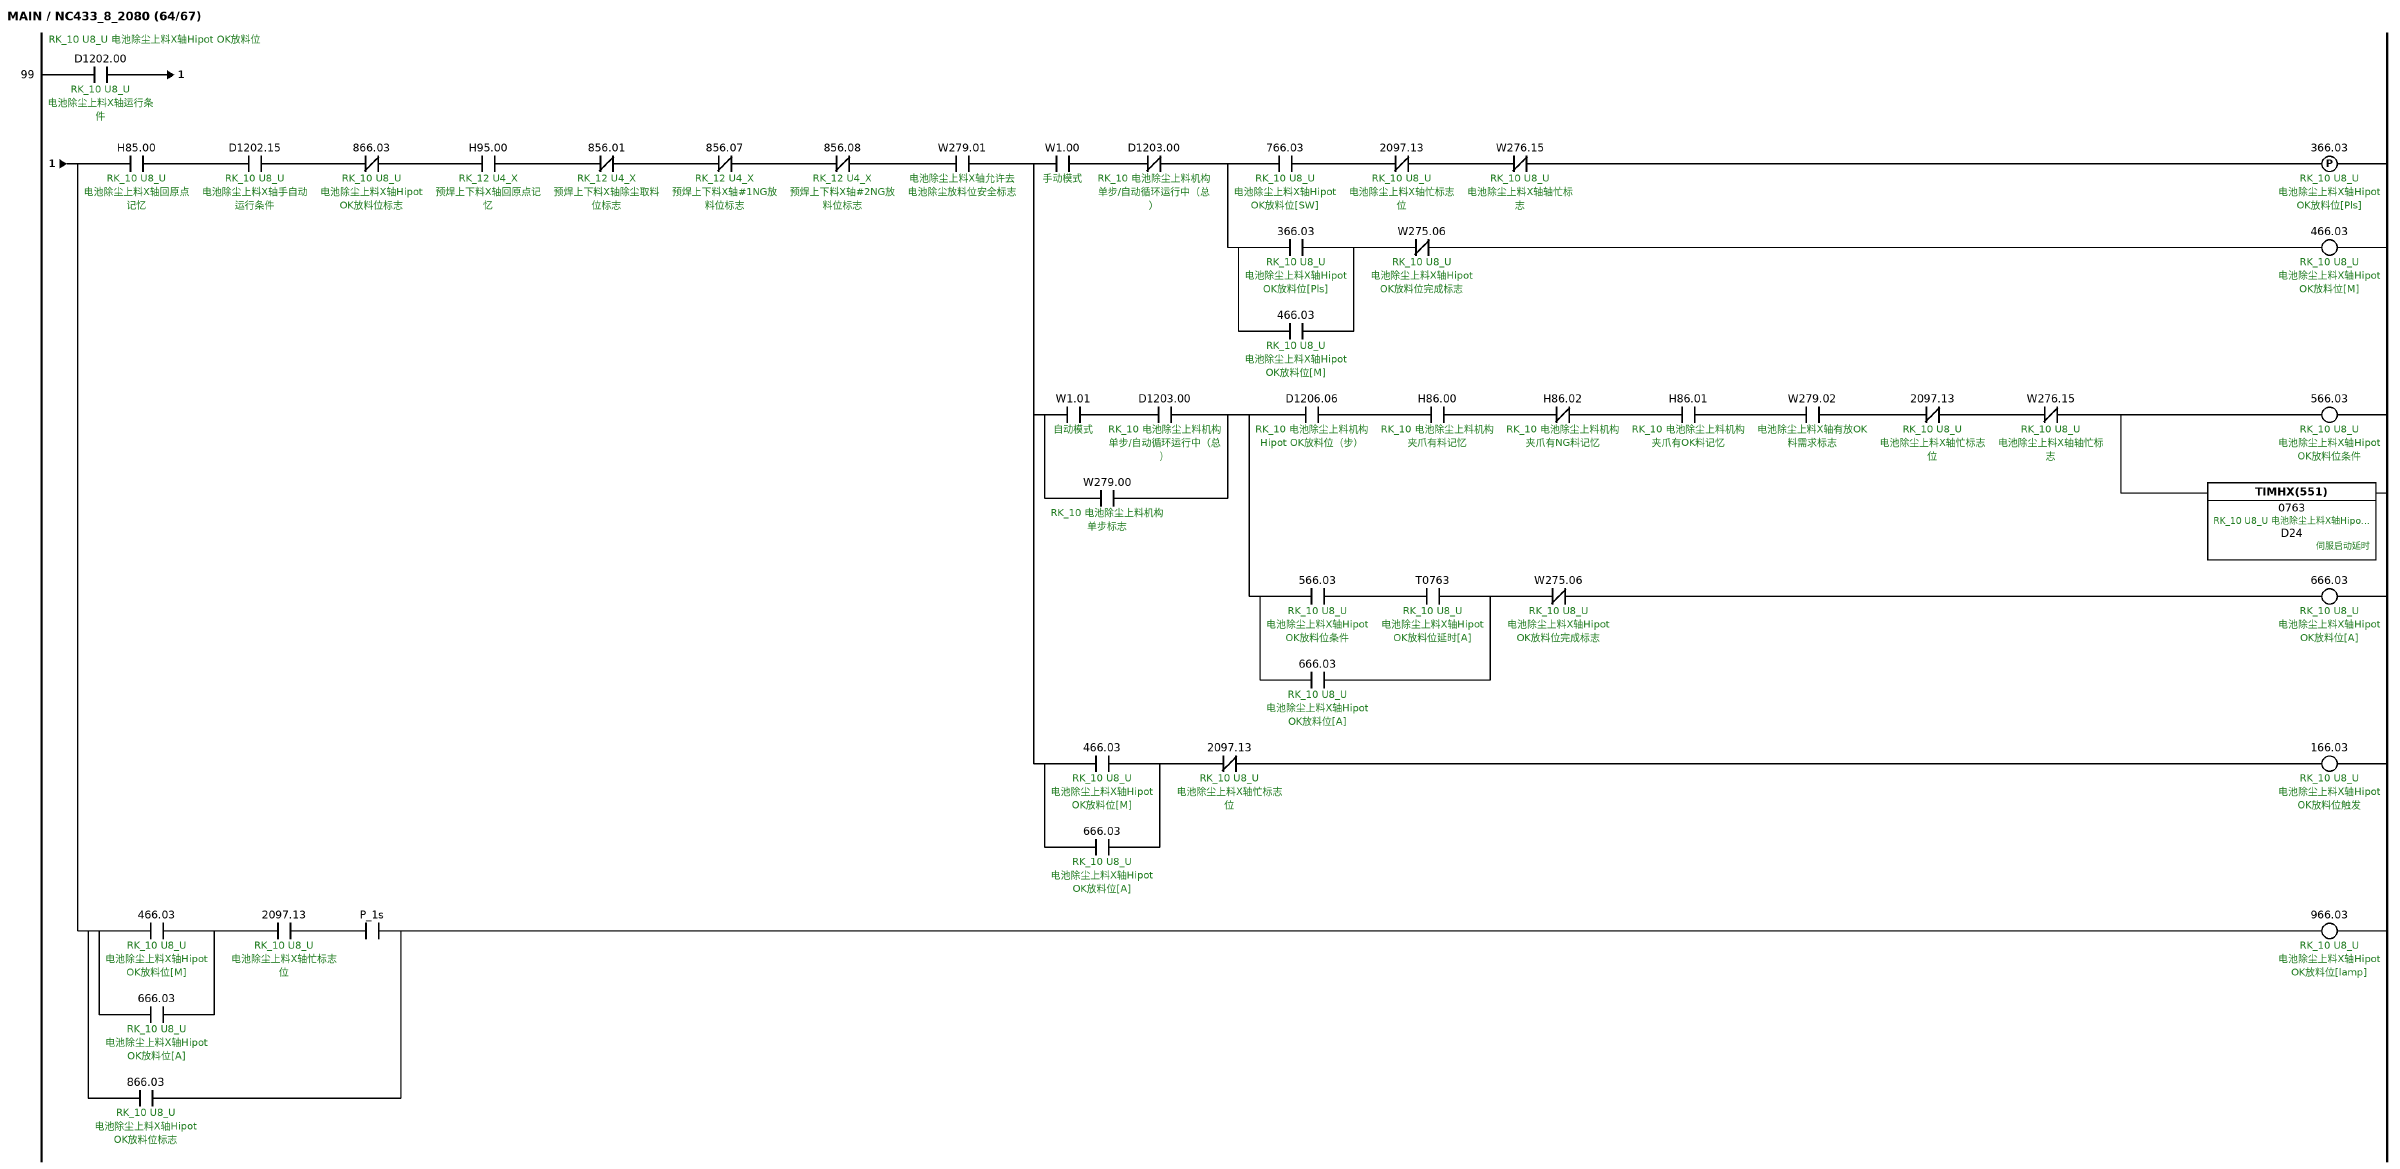
; rung 99: RK_10 U8_U 电池除尘上料X轴Hipot OK放料位
LD D1202.00  ; RK_10 U8_U 电池除尘上料X轴运行条件
OUT TR0
AND H85.00  ; RK_10 U8_U 电池除尘上料X轴回原点记忆
AND D1202.15  ; RK_10 U8_U 电池除尘上料X轴手自动运行条件
ANDNOT 866.03  ; RK_10 U8_U 电池除尘上料X轴Hipot OK放料位标志
AND H95.00  ; RK_12 U4_X 预焊上下料X轴回原点记忆
ANDNOT 856.01  ; RK_12 U4_X 预焊上下料X轴除尘取料位标志
ANDNOT 856.07  ; RK_12 U4_X 预焊上下料X轴#1NG放料位标志
ANDNOT 856.08  ; RK_12 U4_X 预焊上下料X轴#2NG放料位标志
AND W279.01  ; 电池除尘上料X轴允许去电池除尘放料位安全标志
OUT TR1
AND W1.00  ; 手动模式
ANDNOT D1203.00  ; RK_10 电池除尘上料机构单步/自动循环运行中（总）
OUT TR2
AND 766.03  ; RK_10 U8_U 电池除尘上料X轴Hipot OK放料位[SW]
ANDNOT 2097.13  ; RK_10 U8_U 电池除尘上料X轴忙标志位
ANDNOT W276.15  ; RK_10 U8_U 电池除尘上料X轴轴忙标志
DIFU(013) 366.03  ; RK_10 U8_U 电池除尘上料X轴Hipot OK放料位[Pls]
LD TR2
LD 366.03  ; RK_10 U8_U 电池除尘上料X轴Hipot OK放料位[Pls]
OR 466.03  ; RK_10 U8_U 电池除尘上料X轴Hipot OK放料位[M]
ANDLD
ANDNOT W275.06  ; RK_10 U8_U 电池除尘上料X轴Hipot OK放料位完成标志
OUT 466.03  ; RK_10 U8_U 电池除尘上料X轴Hipot OK放料位[M]
LD TR1
LD W1.01  ; 自动模式
AND D1203.00  ; RK_10 电池除尘上料机构单步/自动循环运行中（总）
OR W279.00  ; RK_10 电池除尘上料机构单步标志
ANDLD
OUT TR2
AND D1206.06  ; RK_10 电池除尘上料机构Hipot OK放料位（步）
AND H86.00  ; RK_10 电池除尘上料机构夹爪有料记忆
ANDNOT H86.02  ; RK_10 电池除尘上料机构夹爪有NG料记忆
AND H86.01  ; RK_10 电池除尘上料机构夹爪有OK料记忆
AND W279.02  ; 电池除尘上料X轴有放OK料需求标志
ANDNOT 2097.13  ; RK_10 U8_U 电池除尘上料X轴忙标志位
ANDNOT W276.15  ; RK_10 U8_U 电池除尘上料X轴轴忙标志
OUT 566.03  ; RK_10 U8_U 电池除尘上料X轴Hipot OK放料位条件
TIMHX(551) 0763 D24  ; 伺服启动延时, RK_10 U8_U 电池除尘上料X轴Hipot OK放料位延时[A]
LD TR2
LD 566.03  ; RK_10 U8_U 电池除尘上料X轴Hipot OK放料位条件
AND T0763  ; RK_10 U8_U 电池除尘上料X轴Hipot OK放料位延时[A]
OR 666.03  ; RK_10 U8_U 电池除尘上料X轴Hipot OK放料位[A]
ANDLD
ANDNOT W275.06  ; RK_10 U8_U 电池除尘上料X轴Hipot OK放料位完成标志
OUT 666.03  ; RK_10 U8_U 电池除尘上料X轴Hipot OK放料位[A]
LD TR1
LD 466.03  ; RK_10 U8_U 电池除尘上料X轴Hipot OK放料位[M]
OR 666.03  ; RK_10 U8_U 电池除尘上料X轴Hipot OK放料位[A]
ANDLD
ANDNOT 2097.13  ; RK_10 U8_U 电池除尘上料X轴忙标志位
OUT 166.03  ; RK_10 U8_U 电池除尘上料X轴Hipot OK放料位触发
LD TR0
LD 466.03  ; RK_10 U8_U 电池除尘上料X轴Hipot OK放料位[M]
OR 666.03  ; RK_10 U8_U 电池除尘上料X轴Hipot OK放料位[A]
AND 2097.13  ; RK_10 U8_U 电池除尘上料X轴忙标志位
AND P_1s
OR 866.03  ; RK_10 U8_U 电池除尘上料X轴Hipot OK放料位标志
ANDLD
OUT 966.03  ; RK_10 U8_U 电池除尘上料X轴Hipot OK放料位[lamp]

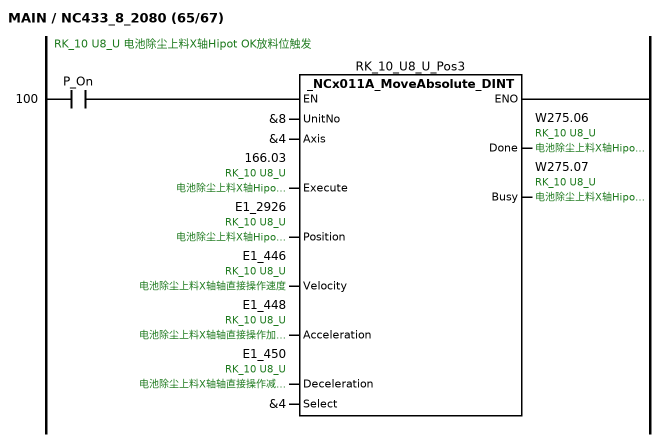
; rung 100: RK_10 U8_U 电池除尘上料X轴Hipot OK放料位触发
LD P_On
CALL RK_10_U8_U_Pos3 : _NCx011A_MoveAbsolute_DINT (UnitNo := &8, Axis := &4, Execute := 166.03, Position := E1_2926, Velocity := E1_446, Acceleration := E1_448, Deceleration := E1_450, Select := &4, Done => W275.06, Busy => W275.07)  ; RK_10 U8_U 电池除尘上料X轴Hipot OK放料位触发, RK_10 U8_U 电池除尘上料X轴Hipot OK放料位, RK_10 U8_U 电池除尘上料X轴轴直接操作速度, RK_10 U8_U 电池除尘上料X轴轴直接操作加速时间, RK_10 U8_U 电池除尘上料X轴轴直接操作减速时间, RK_10 U8_U 电池除尘上料X轴Hipot OK放料位完成标志, RK_10 U8_U 电池除尘上料X轴Hipot OK放料位忙标志

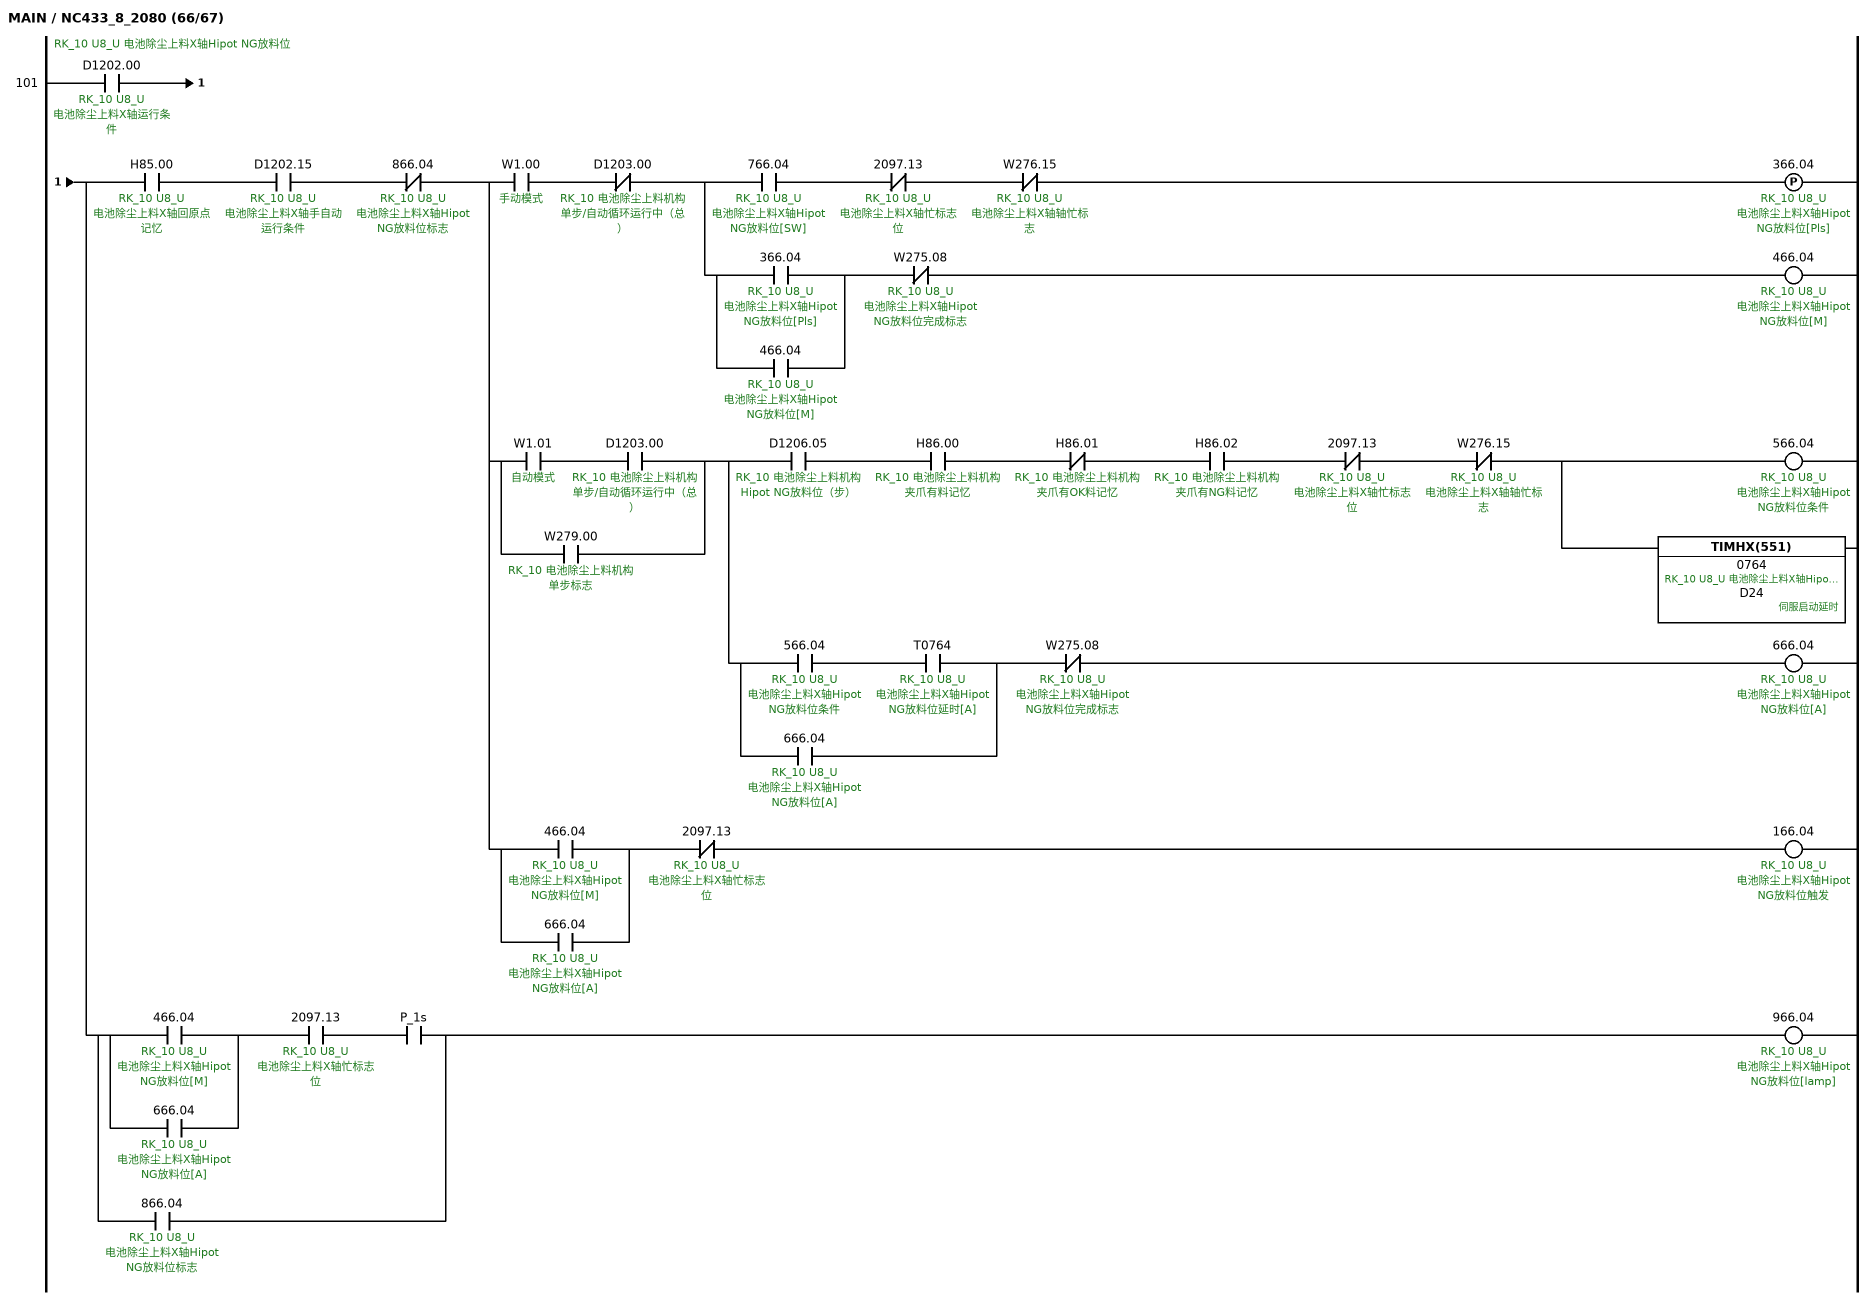
; rung 101: RK_10 U8_U 电池除尘上料X轴Hipot NG放料位
LD D1202.00  ; RK_10 U8_U 电池除尘上料X轴运行条件
OUT TR0
AND H85.00  ; RK_10 U8_U 电池除尘上料X轴回原点记忆
AND D1202.15  ; RK_10 U8_U 电池除尘上料X轴手自动运行条件
ANDNOT 866.04  ; RK_10 U8_U 电池除尘上料X轴Hipot NG放料位标志
OUT TR1
AND W1.00  ; 手动模式
ANDNOT D1203.00  ; RK_10 电池除尘上料机构单步/自动循环运行中（总）
OUT TR2
AND 766.04  ; RK_10 U8_U 电池除尘上料X轴Hipot NG放料位[SW]
ANDNOT 2097.13  ; RK_10 U8_U 电池除尘上料X轴忙标志位
ANDNOT W276.15  ; RK_10 U8_U 电池除尘上料X轴轴忙标志
DIFU(013) 366.04  ; RK_10 U8_U 电池除尘上料X轴Hipot NG放料位[Pls]
LD TR2
LD 366.04  ; RK_10 U8_U 电池除尘上料X轴Hipot NG放料位[Pls]
OR 466.04  ; RK_10 U8_U 电池除尘上料X轴Hipot NG放料位[M]
ANDLD
ANDNOT W275.08  ; RK_10 U8_U 电池除尘上料X轴Hipot NG放料位完成标志
OUT 466.04  ; RK_10 U8_U 电池除尘上料X轴Hipot NG放料位[M]
LD TR1
LD W1.01  ; 自动模式
AND D1203.00  ; RK_10 电池除尘上料机构单步/自动循环运行中（总）
OR W279.00  ; RK_10 电池除尘上料机构单步标志
ANDLD
OUT TR2
AND D1206.05  ; RK_10 电池除尘上料机构Hipot NG放料位（步）
AND H86.00  ; RK_10 电池除尘上料机构夹爪有料记忆
ANDNOT H86.01  ; RK_10 电池除尘上料机构夹爪有OK料记忆
AND H86.02  ; RK_10 电池除尘上料机构夹爪有NG料记忆
ANDNOT 2097.13  ; RK_10 U8_U 电池除尘上料X轴忙标志位
ANDNOT W276.15  ; RK_10 U8_U 电池除尘上料X轴轴忙标志
OUT 566.04  ; RK_10 U8_U 电池除尘上料X轴Hipot NG放料位条件
TIMHX(551) 0764 D24  ; 伺服启动延时, RK_10 U8_U 电池除尘上料X轴Hipot NG放料位延时[A]
LD TR2
LD 566.04  ; RK_10 U8_U 电池除尘上料X轴Hipot NG放料位条件
AND T0764  ; RK_10 U8_U 电池除尘上料X轴Hipot NG放料位延时[A]
OR 666.04  ; RK_10 U8_U 电池除尘上料X轴Hipot NG放料位[A]
ANDLD
ANDNOT W275.08  ; RK_10 U8_U 电池除尘上料X轴Hipot NG放料位完成标志
OUT 666.04  ; RK_10 U8_U 电池除尘上料X轴Hipot NG放料位[A]
LD TR1
LD 466.04  ; RK_10 U8_U 电池除尘上料X轴Hipot NG放料位[M]
OR 666.04  ; RK_10 U8_U 电池除尘上料X轴Hipot NG放料位[A]
ANDLD
ANDNOT 2097.13  ; RK_10 U8_U 电池除尘上料X轴忙标志位
OUT 166.04  ; RK_10 U8_U 电池除尘上料X轴Hipot NG放料位触发
LD TR0
LD 466.04  ; RK_10 U8_U 电池除尘上料X轴Hipot NG放料位[M]
OR 666.04  ; RK_10 U8_U 电池除尘上料X轴Hipot NG放料位[A]
AND 2097.13  ; RK_10 U8_U 电池除尘上料X轴忙标志位
AND P_1s
OR 866.04  ; RK_10 U8_U 电池除尘上料X轴Hipot NG放料位标志
ANDLD
OUT 966.04  ; RK_10 U8_U 电池除尘上料X轴Hipot NG放料位[lamp]

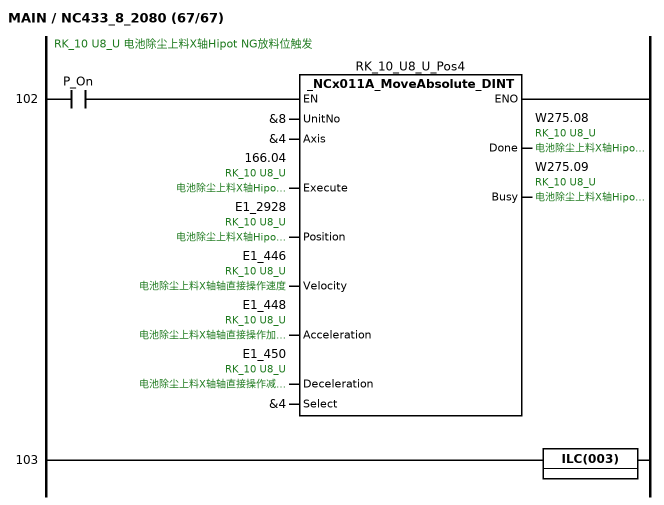
; rung 102: RK_10 U8_U 电池除尘上料X轴Hipot NG放料位触发
LD P_On
CALL RK_10_U8_U_Pos4 : _NCx011A_MoveAbsolute_DINT (UnitNo := &8, Axis := &4, Execute := 166.04, Position := E1_2928, Velocity := E1_446, Acceleration := E1_448, Deceleration := E1_450, Select := &4, Done => W275.08, Busy => W275.09)  ; RK_10 U8_U 电池除尘上料X轴Hipot NG放料位触发, RK_10 U8_U 电池除尘上料X轴Hipot NG放料位, RK_10 U8_U 电池除尘上料X轴轴直接操作速度, RK_10 U8_U 电池除尘上料X轴轴直接操作加速时间, RK_10 U8_U 电池除尘上料X轴轴直接操作减速时间, RK_10 U8_U 电池除尘上料X轴Hipot NG放料位完成标志, RK_10 U8_U 电池除尘上料X轴Hipot NG放料位忙标志
; rung 103
ILC(003)

### Section 入壳压力计算

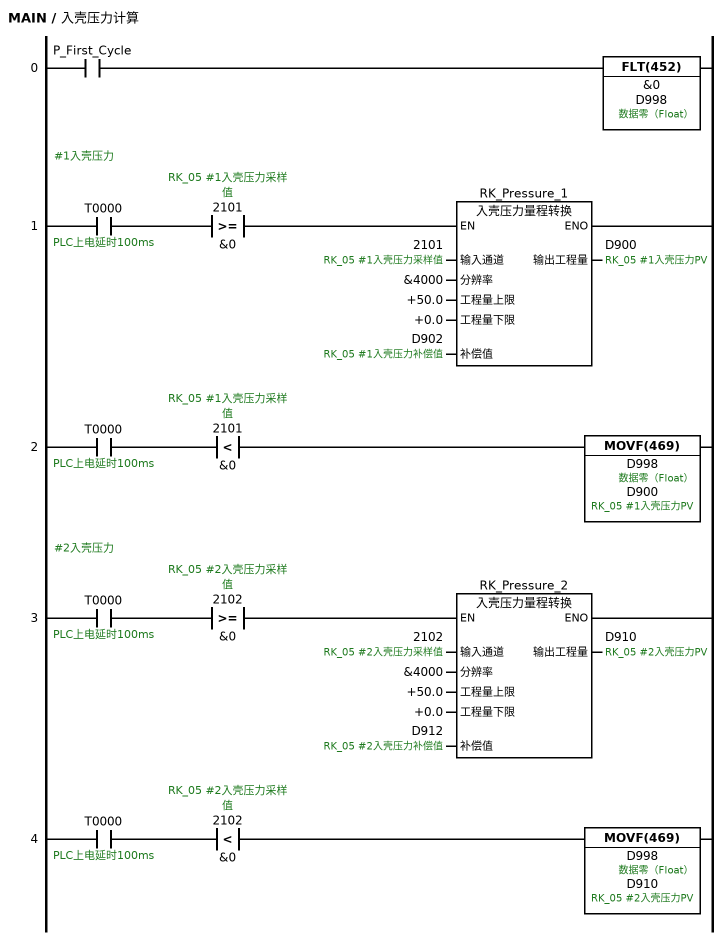
; rung 0
LD P_First_Cycle
FLT(452) &0 D998  ; 数据零（Float）
; rung 1: #1入壳压力
LD T0000  ; PLC上电延时100ms
AND>=S(327) 2101 &0  ; RK_05 #1入壳压力采样值
CALL RK_Pressure_1 : 入壳压力量程转换 (输入通道 := 2101, 分辨率 := &4000, 工程量上限 := +50.0, 工程量下限 := +0.0, 补偿值 := D902, 输出工程量 => D900)  ; RK_05 #1入壳压力采样值, RK_05 #1入壳压力补偿值, RK_05 #1入壳压力PV
; rung 2
LD T0000  ; PLC上电延时100ms
AND<S(312) 2101 &0  ; RK_05 #1入壳压力采样值
MOVF(469) D998 D900  ; 数据零（Float）, RK_05 #1入壳压力PV
; rung 3: #2入壳压力
LD T0000  ; PLC上电延时100ms
AND>=S(327) 2102 &0  ; RK_05 #2入壳压力采样值
CALL RK_Pressure_2 : 入壳压力量程转换 (输入通道 := 2102, 分辨率 := &4000, 工程量上限 := +50.0, 工程量下限 := +0.0, 补偿值 := D912, 输出工程量 => D910)  ; RK_05 #2入壳压力采样值, RK_05 #2入壳压力补偿值, RK_05 #2入壳压力PV
; rung 4
LD T0000  ; PLC上电延时100ms
AND<S(312) 2102 &0  ; RK_05 #2入壳压力采样值
MOVF(469) D998 D910  ; 数据零（Float）, RK_05 #2入壳压力PV

### Section 复位

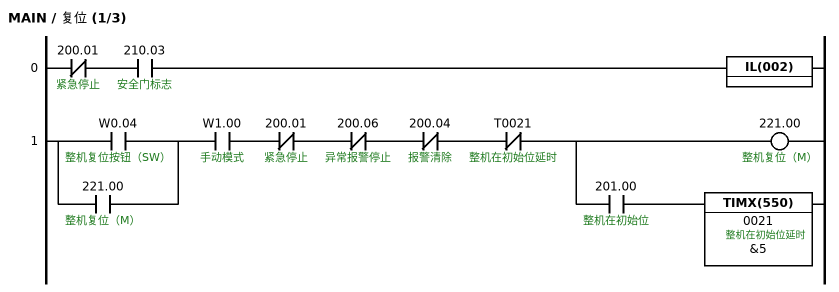
; rung 0
LDNOT 200.01  ; 紧急停止
AND 210.03  ; 安全门标志
IL(002)
; rung 1
LD W0.04  ; 整机复位按钮（SW）
OR 221.00  ; 整机复位（M）
AND W1.00  ; 手动模式
ANDNOT 200.01  ; 紧急停止
ANDNOT 200.06  ; 异常报警停止
ANDNOT 200.04  ; 报警清除
ANDNOT T0021  ; 整机在初始位延时
OUT 221.00  ; 整机复位（M）
AND 201.00  ; 整机在初始位
TIMX(550) 0021 &5  ; 整机在初始位延时

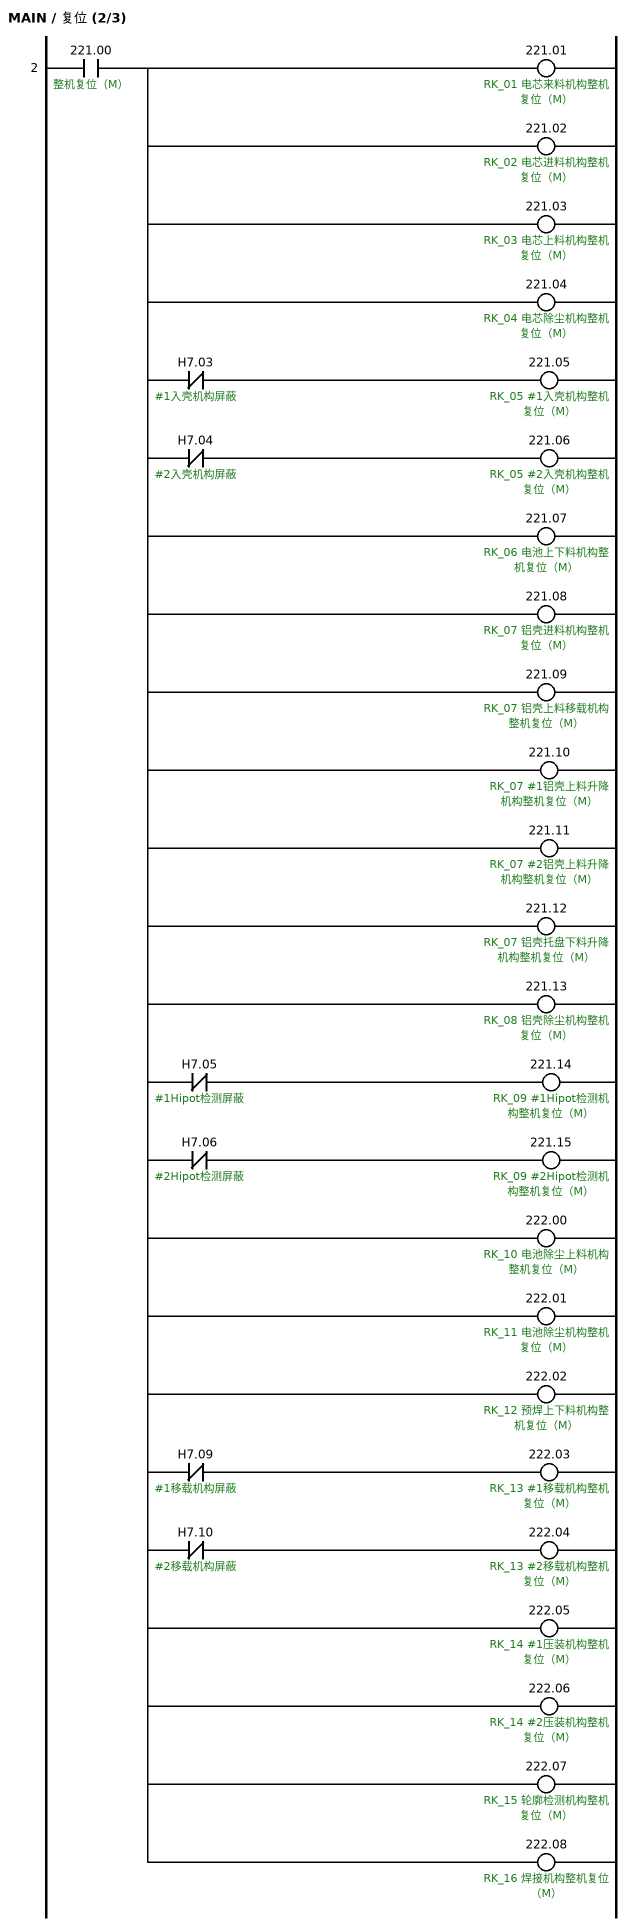
; rung 2
LD 221.00  ; 整机复位（M）
OUT TR0
OUT 221.01  ; RK_01 电芯来料机构整机复位（M）
OUT 221.02  ; RK_02 电芯进料机构整机复位（M）
OUT 221.03  ; RK_03 电芯上料机构整机复位（M）
OUT 221.04  ; RK_04 电芯除尘机构整机复位（M）
ANDNOT H7.03  ; #1入壳机构屏蔽
OUT 221.05  ; RK_05 #1入壳机构整机复位（M）
LD TR0
ANDNOT H7.04  ; #2入壳机构屏蔽
OUT 221.06  ; RK_05 #2入壳机构整机复位（M）
LD TR0
OUT 221.07  ; RK_06 电池上下料机构整机复位（M）
OUT 221.08  ; RK_07 铝壳进料机构整机复位（M）
OUT 221.09  ; RK_07 铝壳上料移载机构整机复位（M）
OUT 221.10  ; RK_07 #1铝壳上料升降机构整机复位（M）
OUT 221.11  ; RK_07 #2铝壳上料升降机构整机复位（M）
OUT 221.12  ; RK_07 铝壳托盘下料升降机构整机复位（M）
OUT 221.13  ; RK_08 铝壳除尘机构整机复位（M）
ANDNOT H7.05  ; #1Hipot检测屏蔽
OUT 221.14  ; RK_09 #1Hipot检测机构整机复位（M）
LD TR0
ANDNOT H7.06  ; #2Hipot检测屏蔽
OUT 221.15  ; RK_09 #2Hipot检测机构整机复位（M）
LD TR0
OUT 222.00  ; RK_10 电池除尘上料机构整机复位（M）
OUT 222.01  ; RK_11 电池除尘机构整机复位（M）
OUT 222.02  ; RK_12 预焊上下料机构整机复位（M）
ANDNOT H7.09  ; #1移载机构屏蔽
OUT 222.03  ; RK_13 #1移载机构整机复位（M）
LD TR0
ANDNOT H7.10  ; #2移载机构屏蔽
OUT 222.04  ; RK_13 #2移载机构整机复位（M）
LD TR0
OUT 222.05  ; RK_14 #1压装机构整机复位（M）
OUT 222.06  ; RK_14 #2压装机构整机复位（M）
OUT 222.07  ; RK_15 轮廓检测机构整机复位（M）
OUT 222.08  ; RK_16 焊接机构整机复位（M）

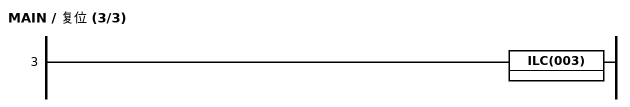
; rung 3
ILC(003)

### Section 指示灯

